    // Vị trí Conveyor hiện tại dùng cho giám sát.
    CurrentConveyorPositionMM : LREAL;
	
	CaptureConveyorPos      : REAL;     // Position conveyor lúc chụp.
	
	CaptureRobotPos         : ST_POS;   // Position robot lúc chụp.

    VisionPos               : ST_POS;   // Position vision trả về.

    // Điểm Score của Vision.
    // Với Sensor có thể gán mặc định 100%.
    VisionScore : REAL;

    // TRUE nếu góc Object có giá trị tin cậy.
    OrientationValid : BOOL;
	
// 	// TRUE khi Object Vision đã có kết quả Pose hợp lệ.
// 	VisionResultValid : BOOL;

    // TRUE khi Object đã được một Tool giữ chỗ.
    Reserved : BOOL;

    // ToolID đang giữ Object.
    ReservedToolID : UINT;

    // Trạng thái Object.
    State : E_TrackingObjectState;
	
    TriggerID               : UDINT;    // TriggerID vision.
    ProductID               : UDINT;    // ID sản phẩm.

    CameraID                : UINT;     // Camera đã chụp.
    JobID                   : UINT;     // Job đã sử dụng.

    

    ConveyorOffset          : REAL;     // Conveyor dịch từ lúc chụp.
    ConveyorCoordinate      : REAL;     // Tọa độ dọc conveyor hiện tại.

    CurrentPos              : ST_POS;   // Position hiện tại của object.

    InspectionResult        : E_InspectionResult; // Kết quả kiểm tra.
    PickAttempts            : UINT;     // Số lần thử gắp.

    RejectCode              : UINT;     // Mã lý do reject.
    ErrorID                 : UDINT;    // Mã lỗi object.
	
	// TRUE khi object còn đủ thời gian và nằm trong vùng có thể nhận gắp.
    CanPick              : BOOL;

    // Thời gian ước tính còn lại trước khi tới giới hạn bắt đầu gắp, giây.
    TimeRemainingSec     : REAL;

    // TRUE khi object active đã vượt AbortPositionMM.
    AbortRequired        : BOOL;

    // Dùng debug/thống kê lý do object bị bỏ.
    MissCode             : UINT;
	// Mức ưu tiên của object.
    // Giá trị lớn hơn được ưu tiên hơn.
    Priority : UINT;

    // Điểm chất lượng kết quả Vision, thường nằm trong khoảng 0.0 đến 1.0
    // hoặc 0.0 đến 100.0 tùy phần mềm Vision.
    //VisionScore : REAL;

    // Thời gian robot ước tính cần để tiếp cận và gắp object, đơn vị giây.
    // Giai đoạn đầu có thể gán bằng cùng một giá trị cho mọi object.
    EstimatedPickTimeSec : REAL;

    // Thời điểm object được thêm vào Queue.
    // Dùng cho thuật toán FIFO.
    CaptureTime : TIME;


END_STRUCT
END_TYPE

// Just_Motion_Control_x86_64_Linux_SM_WV/Application/STRUCT_/ConveyorTracking/ST_TRACKING_QUEUE
TYPE ST_TRACKING_QUEUE :
STRUCT
    Objects             : ARRAY[0..GVL.C_MAX_TRACK_OBJECTS]
                          OF ST_TRACKING_OBJECT;

    ValidCount          : UINT;     // Tổng số object hợp lệ.
    ReservedCount       : UINT;     // Tổng số object đã reserve.

    ActiveIndex         : UINT;     // Index object đang được xử lý.
    NextObjectID        : UDINT;    // Bộ tạo ObjectID tiếp theo.

    LastResult          : E_QueueResult; // Kết quả thao tác queue gần nhất.
END_STRUCT
END_TYPE

// Just_Motion_Control_x86_64_Linux_SM_WV/Application/STRUCT_/ConveyorTracking/ST_TRACKING_RUNTIME
TYPE ST_TRACKING_RUNTIME :
STRUCT
    State               : E_TrackingState;     // Trạng thái manager.
    Request             : ST_MODULE_REQUEST;
    Response            : ST_MODULE_RESPONSE;

    SelectedObjectIndex : UINT;                // Index object đã chọn.
    SelectedObjectID    : UDINT;               // ID object đã chọn.

    ApproachPos         : ST_POS;              // Điểm approach trong PCS.
    PickPos             : ST_POS;              // Điểm pick trong PCS.
    RetractPos          : ST_POS;              // Điểm retract trong PCS.

    PCSInfo             : ST_PCS_INFO;         // Dữ liệu PCS hiện tại.

    PickSuccess         : BOOL;                // TRUE khi gắp thành công.
    ErrorInfo           : ST_ERROR_INFO;       // Thông tin lỗi.
END_STRUCT
END_TYPE

// Just_Motion_Control_x86_64_Linux_SM_WV/Application/STRUCT_/ConveyorTracking/ST_TRACKING_SIMULATION_CONFIG
TYPE ST_TRACKING_SIMULATION_CONFIG :
STRUCT
	Mode : E_ApplicationSimulationMode;

    // Encoder ảo.
    VirtualEncoderEnable : BOOL;
    VirtualEncoderReset : BOOL;
    VirtualEncoderStepPerCycle : DINT;

    // Object giả.
    FixedObjectEnable : BOOL;
    FixedObjectPosition : MC_COORD_REF;

    // Vacuum giả.
    AutoVacuumOK : BOOL;
    VacuumOKDelay : TIME;

    // Motion logic-only.
    LogicMotionDuration : TIME;

    // Cho phép dừng sau từng state để debug.
    SingleStateMode : BOOL;
    ContinueState : BOOL;

END_STRUCT
END_TYPE

// Just_Motion_Control_x86_64_Linux_SM_WV/Application/STRUCT_/ConveyorTracking/ST_TRACKING_WORKSPACE_CONFIG
TYPE ST_TRACKING_WORKSPACE_CONFIG :
STRUCT
	// Vị trí bắt đầu vùng thu nhận object, đơn vị mm.
    AcquireZoneStartMM : REAL;

    // Vị trí bắt đầu vùng được phép gắp, đơn vị mm.
    PickZoneStartMM : REAL;

    // Vị trí kết thúc vùng được phép gắp, đơn vị mm.
    PickZoneEndMM : REAL;

    // Vượt vị trí này mà chưa VacuumOK thì phải bỏ object active.
    AbortPositionMM : REAL;

    // Vượt vị trí này thì object chưa active bị EXPIRED.
    ExpirePositionMM : REAL;

//     // Khoảng cách tối thiểu mong muốn giữa hai object, đơn vị mm.
//     MinimumObjectSpacingMM : REAL;

    // Thời gian tối thiểu robot cần để thực hiện thao tác gắp, đơn vị giây.
    MinimumPickTimeSec : REAL;

    // Thời gian dự phòng an toàn, đơn vị giây.
    SafetyMarginTimeSec : REAL;
END_STRUCT
END_TYPE

// Just_Motion_Control_x86_64_Linux_SM_WV/Application/STRUCT_/ConveyorTracking/ST_TrackingObjectQueue
//=============================================================================
// DUT: TRACKING OBJECT QUEUE
//=============================================================================
TYPE ST_TrackingObjectQueue :
STRUCT

    // Danh sách Object.
    Objects : ARRAY[0..GVL.C_MAX_TRACK_OBJECTS] OF ST_TRACKING_OBJECT;

    // Số Object đang có trong Queue.
    Count : UINT;

    // Bộ đếm sinh ObjectID cho Sensor Source.
    NextObjectID : UDINT;

END_STRUCT
END_TYPE

// Just_Motion_Control_x86_64_Linux_SM_WV/Application/STRUCT_/ConveyorTracking/ST_VISION_TRACK_OBJECT_ITEM
TYPE ST_VISION_TRACK_OBJECT_ITEM :
STRUCT

    // TRUE khi Object này hợp lệ.
    Valid : BOOL;

    // Tọa độ Object do Vision trả.
    // Có thể là pixel hoặc mm tùy cấu hình Tracking Vision Source.
    Pos : ST_POS;

    // Score nhận dạng.
    Score : REAL;

    // Product Class nếu Vision có phân loại.
    // 0 = sử dụng ProductClassID mặc định của Source Config.
    ProductClassID : UINT;

    // ID do Vision cấp cho Detection nếu có.
    FeatureID : UDINT;

END_STRUCT
END_TYPE

// Just_Motion_Control_x86_64_Linux_SM_WV/Application/STRUCT_/ConveyorTracking/ST_VISION_TRACK_OBJECT_RESULT
TYPE ST_VISION_TRACK_OBJECT_RESULT :
STRUCT

    // TRUE khi toàn bộ danh sách Object hợp lệ.
    Valid : BOOL;

    // Số Object thực Vision trả.
    ObjectCount : UINT;

    // Danh sách Object.
    Objects :
        ARRAY[1..GVL.C_MAX_VISION_TRACK_OBJECTS_PER_FRAME]
        OF ST_VISION_TRACK_OBJECT_ITEM;

END_STRUCT
END_TYPE

// Just_Motion_Control_x86_64_Linux_SM_WV/Application/STRUCT_/ConveyorTracking/ST_VisionTrackingDetection
TYPE ST_VisionTrackingDetection :
STRUCT

    // Detection này hợp lệ.
    Valid : BOOL;

    // Pose raw Vision trả về.
    RawPos : ST_POS;

    // Score.
    Score : REAL;

    // Product Class do Vision trả.
    // 0 = dùng ProductClassID trong Config.
    ProductClassID : UINT;

    // Feature/Object ID nếu Vision có.
    FeatureID : UDINT;

END_STRUCT
END_TYPE

// Just_Motion_Control_x86_64_Linux_SM_WV/Application/STRUCT_/ConveyorTracking/ST_VisionTrackingMultiResult
TYPE ST_VisionTrackingMultiResult :
STRUCT

    // Bộ kết quả hoàn chỉnh.
    Valid : BOOL;

    // Trigger tương ứng frame ảnh.
    TriggerID : UDINT;

    // Camera.
    CameraID : UINT;

    // Job.
    JobID : UINT;

    // Vị trí Conveyor tại đúng lúc chụp ảnh.
    CaptureConveyorPositionMM : LREAL;

    // Số Object Vision tìm thấy.
    ObjectCount : UINT;

    // Danh sách Detection.
    Objects :
        ARRAY[1..GVL.C_MAX_VISION_TRACK_OBJECTS_PER_FRAME]
        OF ST_VisionTrackingDetection;

END_STRUCT
END_TYPE

// Just_Motion_Control_x86_64_Linux_SM_WV/Application/STRUCT_/ConveyorTracking/ST_VisionTrackingSourceConfig
//=============================================================================
// DUT: ST_VisionTrackingSourceConfig
//-----------------------------------------------------------------------------
// Cấu hình một nguồn Vision dùng để tạo Object cho Conveyor Tracking.
// Đây là BẢN THAY THẾ cho DUT hiện tại: giữ toàn bộ field cũ và bổ sung phần
// BACKGROUND TRIGGER ở cuối.
//=============================================================================
TYPE ST_VisionTrackingSourceConfig :
STRUCT

    //=========================================================================
    // SOURCE IDENTITY
    //=========================================================================
    Enable : BOOL;                          // TRUE = cho phép Source hoạt động.
    VisionSourceID : UINT;                  // ID duy nhất của nguồn Vision Tracking.
    VisionSourceName : STRING[32];          // Tên hiển thị trên HMI/debug.
    CameraID : UINT;                        // Camera dùng cho Source này.
    JobID : UINT;                           // Job Vision dùng để tìm Object.

    //=========================================================================
    // PRODUCT / FILTER
    //=========================================================================
    ProductClassID : UINT;                  // Class mặc định nếu Vision trả ProductClassID = 0.
    MinimumScore : REAL;                    // Object có Score thấp hơn giá trị này sẽ bị loại.
    MaxObjectCount : UINT;                  // Số Object tối đa nhận từ một frame.

    //=========================================================================
    // SCALE VISION
    //-------------------------------------------------------------------------
    // ResultInPixel = TRUE:
    //     X/Y raw của Vision được đổi pixel -> mm bằng MMPerPixelX/Y.
    // ResultInPixel = FALSE:
    //     X/Y được coi là mm; nên đặt MMPerPixelX/Y = 1.0 để dễ theo dõi.
    //=========================================================================
    ResultInPixel : BOOL;
    MMPerPixelX : REAL;
    MMPerPixelY : REAL;

    //=========================================================================
    // VISION OFFSET
    //-------------------------------------------------------------------------
    // Fine offset sau khi kết quả Vision đã được chuẩn hóa về Conveyor CS.
    // Không dùng field này thay cho Tool PickOffset hoặc Product Height.
    //=========================================================================
    VisionOffset : ST_POS;

    //=========================================================================
    // DUPLICATE FILTER
    //-------------------------------------------------------------------------
    // Dùng để so Object mới với Object đang có trong Tracking Queue.
    // Object RESERVED/TRACKING/PICKING vẫn phải được xét duplicate vì Camera
    // có thể nhìn lại đúng Object đang được Robot xử lý.
    //=========================================================================
    DuplicateToleranceXMM : REAL;
    DuplicateToleranceYMM : REAL;
    DuplicateAngleDeg : REAL;

    //=========================================================================
    // BACKGROUND CAMERA TRIGGER - NEW
    //-------------------------------------------------------------------------
    // Tracking Vision không trigger trong TRK_PICK/TRK_CREATE_PCS.
    // Source này chạy nền trong thời gian TRACK_PICK session đang active.
    //=========================================================================
    AutoTrigger : BOOL;                     // TRUE = tự trigger theo quãng đường Conveyor.
    TriggerPitchMM : REAL;                  // Conveyor đi thêm bao nhiêu mm thì phát frame mới.
    TriggerOnlyWhenMoving : BOOL;           // TRUE = chỉ trigger khi Conveyor đang chạy.
    MinimumTriggerVelocityMMs : REAL;        // Ngưỡng tốc độ coi là Conveyor đang chạy.

END_STRUCT
END_TYPE

// Just_Motion_Control_x86_64_Linux_SM_WV/Application/STRUCT_/Geometry/ST_CIRCLE_2D
TYPE ST_CIRCLE_2D :
STRUCT
    CenterPos   : ST_POS;   // Tâm đường tròn.
    Radius      : REAL;     // Bán kính, mm.
    Valid       : BOOL;     // Dữ liệu hình tròn hợp lệ.
END_STRUCT
END_TYPE

// Just_Motion_Control_x86_64_Linux_SM_WV/Application/STRUCT_/Geometry/ST_LINE_2D
TYPE ST_LINE_2D :
STRUCT
    StartPos    : ST_POS;   // Điểm đầu đoạn thẳng.
    EndPos      : ST_POS;   // Điểm cuối đoạn thẳng.
    Valid       : BOOL;     // Đoạn thẳng hợp lệ.
END_STRUCT
END_TYPE

// Just_Motion_Control_x86_64_Linux_SM_WV/Application/STRUCT_/Geometry/ST_PATH_BLOCK
TYPE ST_PATH_BLOCK :
STRUCT
    Valid           : BOOL;     // Block hợp lệ.
    PathID          : UDINT;    // ID đường chạy.

    BlockIndex      : UINT;     // Số thứ tự block.
    BlockCount      : UINT;     // Tổng số block.

    StartPointIndex : UINT;     // Index điểm đầu trong toàn bộ path.
    PointCount      : UINT;     // Số điểm trong block.

    Points          : ARRAY[0..GVL.C_MAX_PATH_BLOCK_POINTS]
                      OF ST_PATH_POINT;

    Checksum        : UDINT;    // Checksum block.
END_STRUCT
END_TYPE

// Just_Motion_Control_x86_64_Linux_SM_WV/Application/STRUCT_/Geometry/ST_PATH_DATA
TYPE ST_PATH_DATA :
STRUCT
    Valid               : BOOL;     // Path hợp lệ.
    Complete            : BOOL;     // Đã nhận đầy đủ dữ liệu.
    Processed           : BOOL;     // Path đã qua xử lý.

    PathID              : UDINT;    // ID đường chạy.
    CoordSystem         : E_AppCoordSystem; // Hệ tọa độ của path.

    RawPointCount       : UINT;     // Số điểm vision trả về.
    ProcessPointCount   : UINT;     // Số điểm sau xử lý.

    ClosedPath          : BOOL;     // TRUE khi là đường khép kín.

    RawPoints           : ARRAY[0..GVL.C_MAX_RAW_PATH_POINTS]
                          OF ST_PATH_POINT;

    ProcessPoints       : ARRAY[0..GVL.C_MAX_PROCESS_PATH_POINTS]
                          OF ST_PATH_POINT;
END_STRUCT
END_TYPE

// Just_Motion_Control_x86_64_Linux_SM_WV/Application/STRUCT_/Geometry/ST_PATH_POINT
TYPE ST_PATH_POINT :
STRUCT
    Valid           : BOOL;                 // Điểm được sử dụng.
    Index           : UINT;                 // Thứ tự điểm.

    Pos             : ST_POS;               // Tọa độ X/Y/Z/A.
    SegmentType     : E_PathSegmentType;    // Kiểu đoạn dẫn tới điểm này.

    GlueOn          : BOOL;                 // TRUE khi cần mở keo trên đoạn.
    Speed           : REAL;                 // Tốc độ đoạn, mm/s.
    Flow            : REAL;                 // Lưu lượng keo.
    BlendRadius     : REAL;                 // Bán kính blend, mm.

    FeatureID       : UINT;                 // ID đoạn vision trả về.
END_STRUCT
END_TYPE

// Just_Motion_Control_x86_64_Linux_SM_WV/Application/STRUCT_/Glue/ST_GLUE_CONFIG
TYPE ST_GLUE_CONFIG :
STRUCT
    Enable                  : BOOL;     // Cho phép chức năng bôi keo.
    RunMode                 : E_GlueRunMode; // Chế độ chạy.

    DefaultSpeed            : REAL;     // Tốc độ mặc định, mm/s.
    DefaultFlow             : REAL;     // Lưu lượng mặc định.

    MinPointDistance        : REAL;     // Khoảng cách điểm nhỏ nhất, mm.
    MaxPointDistance        : REAL;     // Khoảng cách điểm lớn nhất, mm.

    SmoothingEnable         : BOOL;     // Cho phép làm mượt path.
    SmoothingFactor         : REAL;     // Hệ số làm mượt 0...1.

    ApproachHeight          : REAL;     // Độ cao tiếp cận, mm.
    RetractHeight           : REAL;     // Độ cao rút lên, mm.

    PreFlowTime             : TIME;     // Thời gian mở keo trước.
    PostFlowTime            : TIME;     // Thời gian giữ keo cuối path.

    GlueOutput              : UINT;     // Output điều khiển van keo.
END_STRUCT
END_TYPE

// Just_Motion_Control_x86_64_Linux_SM_WV/Application/STRUCT_/Glue/ST_GLUE_RUNTIME
TYPE ST_GLUE_RUNTIME :
STRUCT
    State               : E_GlueState;      // Trạng thái Glue Manager.
    ProcessState        : E_PathProcessState; // Trạng thái xử lý path.

    Request             : ST_MODULE_REQUEST;
    Response            : ST_MODULE_RESPONSE;

    Path                : ST_PATH_DATA;     // Path hiện tại.
    CurrentPointIndex   : UINT;             // Điểm đang được thực hiện.

    GlueOutputState     : BOOL;             // Trạng thái output keo.
    DryRun              : BOOL;             // TRUE khi không bật keo thật.

    ErrorInfo           : ST_ERROR_INFO;    // Thông tin lỗi.
END_STRUCT
END_TYPE

// Just_Motion_Control_x86_64_Linux_SM_WV/Application/STRUCT_/HMI/MainMC
TYPE MainMC :
STRUCT
	Start, Stop, Reset, Man_or_Auto : BOOL;
	yStart, yStop : BOOL;
	yLamp_Yellow, yLamp_Red, yLamp_Green, yBuzz : BOOL;
	AllwayON : BOOL := TRUE;
	AllwayOFF : BOOL := FALSE;
	
	Project_Run : BYTE; // 0 -255 project _0 none
	Mode_Run : BYTE; // 0-255 mode
	Check_Project : BOOL;
	Result_check : BYTE; // 0-none 1 ok 2 nG 3 waiting
	
	Enable_Dynamics_Limit : BOOL;
END_STRUCT
END_TYPE

// Just_Motion_Control_x86_64_Linux_SM_WV/Application/STRUCT_/HMI/MODBUS
TYPE MODBUS :
STRUCT
	en : BOOL;
	iniID : BYTE;
	port	: WORD;
	TCP_UDP	: BOOL;
	DelayRespTime : WORD;
END_STRUCT
END_TYPE

// Just_Motion_Control_x86_64_Linux_SM_WV/Application/STRUCT_/HMI/Project
TYPE Project :
STRUCT
	Project_Run : BYTE; // 0 -255 project _0 none
	Mode_Run : BYTE; // 0-255 mode
	
END_STRUCT
END_TYPE

// Just_Motion_Control_x86_64_Linux_SM_WV/Application/STRUCT_/HMI/TimeRun
TYPE TimeRun :
STRUCT
	Run, Stop , Wait , CLEAR : BOOL;
	Run_S, Run_M, Run_H,
	Stop_S, Stop_M, Stop_H,
	Wait_S, Wait_M, Wait_H,
	Total_S, Total_M, Total_H : WORD;
END_STRUCT
END_TYPE

// Just_Motion_Control_x86_64_Linux_SM_WV/Application/STRUCT_/Modbus/ST_VISION_MODBUS_CONTROL
TYPE ST_VISION_MODBUS_CONTROL :
STRUCT
    RunCalib : BOOL;                                // ControlWord bit2: yêu cầu chạy Calibration.
    CalibPosReady : BOOL;                           // ControlWord bit3: 12 điểm Calibration đã sẵn sàng.
    AckResult : BOOL;                               // ControlWord bit4: PLC đã nhận toàn bộ Result.
    AckBlock : BOOL;                                // ControlWord bit5: PLC đã đọc xong Block hiện tại.
    CalibPointCount : UINT;                         // Số điểm Calibration hợp lệ, tối đa 12.
    RequestBlockIndex : UINT;                       // Block tiếp theo PLC yêu cầu Vision nạp.
    AckBlockIndex : UINT;                           // Block PLC vừa đọc xong.
    CommandCode : UINT;                             // Dự phòng cho Manual/Calibration command.
    CalibrationPoints : ARRAY[1..12] OF ST_POS;     // Chỉ dùng X/Y/A trong mapping Modbus.
END_STRUCT
END_TYPE

// Just_Motion_Control_x86_64_Linux_SM_WV/Application/STRUCT_/Modbus/ST_VISION_MODBUS_STATUS
TYPE ST_VISION_MODBUS_STATUS :
STRUCT
    HeartBeat : BOOL;                               // StatusWord bit0.
    TriggerDone : BOOL;                             // StatusWord bit1.
    CalibDone : BOOL;                               // StatusWord bit2.
    ResultReady : BOOL;                             // StatusWord bit3.
    Busy : BOOL;                                    // StatusWord bit4.
    Run1Slot : BOOL;                                // StatusWord bit5.
    BlockReady : BOOL;                              // StatusWord bit6.
    Error : BOOL;                                   // StatusWord bit7.
    CalibBusy : BOOL;                               // StatusWord bit8.
    CalibError : BOOL;                              // StatusWord bit9.
    BlockIndex : UINT;                              // Block hiện tại trong MultiDataBuffer.
    BlockDataCount : UINT;                          // Số record thực trong Block.
END_STRUCT
END_TYPE

// Just_Motion_Control_x86_64_Linux_SM_WV/Application/STRUCT_/MOTOR/MOTOR_DATA
TYPE MOTOR_DATA :
STRUCT
	POS : ARRAY[0..50] OF REAL;
	SPEED_HIGH, SPEED_MID, SPEED_LOW : REAL;

	MOTION_ACC, MOTION_DEC, MOTION_JERK : REAL;
	LinearDistanceJog, AngularDistanceJog : REAL;
	Fac_Vel, Fac_Acc, Fac_Jerk,Fac_Torque : REAL;
	
	LIMIT_FW, LIMIT_BW: REAL;
END_STRUCT
END_TYPE

// Just_Motion_Control_x86_64_Linux_SM_WV/Application/STRUCT_/MOTOR/MOTOR_IN
TYPE MOTOR_IN :
STRUCT
	Power, Enable, Reset,
	Auto, Manual, Lock,
	HOME, 
	JOG_FW, JOG_BW : BOOL;
	Comfirm_Move, Comfirm_Teach: BOOL;
	LIMIT_FW, LIMIT_BW : LREAL;
	SPEED, ACC, DEC, JERK : REAL;
	Control_w_speed, Control_w_mode : WORD;
END_STRUCT
END_TYPE

// Just_Motion_Control_x86_64_Linux_SM_WV/Application/STRUCT_/MOTOR/MOTOR_OUT
TYPE MOTOR_OUT :
STRUCT
	Ready, Runing, Pause, Stop, 
	ERROR, SAFETY_CHECK : BOOL;
	M_Homed : BOOL;
	CUR_POS: REAL;
	CUR_SP : REAL;
END_STRUCT
END_TYPE

// Just_Motion_Control_x86_64_Linux_SM_WV/Application/STRUCT_/Project/Data_Point_Calib
TYPE Data_Point_Calib :
STRUCT	
	X_POS : ARRAY[0..50] OF REAL;
	Y_POS : ARRAY[0..50] OF REAL;
	Z_POS : ARRAY[0..50] OF REAL;
	R_POS : ARRAY[0..50] OF REAL;
END_STRUCT
END_TYPE

// Just_Motion_Control_x86_64_Linux_SM_WV/Application/STRUCT_/Project/Data_Project_3
TYPE Data_Project_3 :
STRUCT	
	Trigger_Auto, Trigger_Man, Trigger : BOOL; // on chup Cam
	Enable_RB_B, Enable_RB_A : BOOL;
	Shape_T1, Shape_T2 : WORD;
	Data_PlaceB_PickA, Data_PlaceA : ARRAY[0..3] OF WORD;
	
	AllowRB_In_TableC, AllowRB_In_TableA, AllowRB_In_TableB  : WORD; // =0 None : = 1: Allow_RB_B_Place , =2 :Allow_RB_A_Pick 
	
	Pro_A, Pro_B : WORD;
	NextStep_A, NextStep_B, Auto_Man_A, Auto_Man_B : BOOL;
END_STRUCT
END_TYPE

// Just_Motion_Control_x86_64_Linux_SM_WV/Application/STRUCT_/Project/Data_Project
TYPE Data_Project :
STRUCT
	Model_RB_A : ARRAY [0..10] OF Model_Data_RB;
	Model_RB_B : ARRAY [0..10] OF Model_Data_RB;
END_STRUCT
END_TYPE

// Just_Motion_Control_x86_64_Linux_SM_WV/Application/STRUCT_/Project/Project_2
TYPE Project_2 :
STRUCT
	P1,P2,P3,P4 : WORD; // địa chỉ pos
	
	P1_Z,P2_Z,P3_Z,P4_Z : WORD; // số lượng z
	
	pitchZ1, pitchZ2, pitchZ3, pitchZ4 : REAL; // khoảng cách z
	
	P1_Z_,P2_Z_,P3_Z_,P4_Z_  :WORD; // monitor
	
END_STRUCT
END_TYPE

// Just_Motion_Control_x86_64_Linux_SM_WV/Application/STRUCT_/Project/Project_3
TYPE Project_3 :
STRUCT
	
	P1,P2,P3,P4 : WORD; // địa chỉ pos
	
	P1_Z,P2_Z,P3_Z,P4_Z : WORD; // số lượng z
	
	pitchZ1, pitchZ2, pitchZ3, pitchZ4 : REAL; // khoảng cách z
	Delay_T1, Delay_T2 : WORD; 
	
	P1_Z_,P2_Z_,P3_Z_,P4_Z_  :WORD; // monitor
	Target_T1, Target_T2 : ST_POS;
	
	
END_STRUCT
END_TYPE

// Just_Motion_Control_x86_64_Linux_SM_WV/Application/STRUCT_/Project/Project_3_VISION
TYPE Project_3_VISION :
STRUCT
	vis_1, vis_2 : WORD; // địa chỉ pos
	
	Pos_vision_T1, Pos_vision_T1_Offset : ST_POS;
	Pos_vision_T2, Pos_vision_T2_Offset : ST_POS;
	
	Pos_No_T1, Pos_No_T2 : WORD;
	Number_trigger_False : WORD;
	Delay_T1, Delay_T2 : WORD;
	
	Pos_Target_T1, Pos_Target_T2 : ST_POS;
	Status_T1, Status_T2 :WORD;
	
END_STRUCT
END_TYPE

// Just_Motion_Control_x86_64_Linux_SM_WV/Application/STRUCT_/ROBOT/Model_Data_RB_ALL
TYPE Model_Data_RB_ALL :
STRUCT
	DATA_RB_A: RB_DATA;
	DATA_RB_B: RB_DATA;
	Model_Name: STRING[20];
END_STRUCT
END_TYPE

// Just_Motion_Control_x86_64_Linux_SM_WV/Application/STRUCT_/ROBOT/Model_Data_RB
TYPE Model_Data_RB :
STRUCT
	DATA_RB: RB_DATA;
	Model_Name: STRING[20];
END_STRUCT
END_TYPE

// Just_Motion_Control_x86_64_Linux_SM_WV/Application/STRUCT_/ROBOT/Move_Point
TYPE Move_Point :
STRUCT
	Enable	  : BOOL;
	Hand_Type : INT; // o: Trai-A; 1: Phai-B
	Move_Type : INT; // 0: MovP ; 1-MovL; 2-MovC
	A_Error   : BOOL;
	B_Error   : BOOL;
END_STRUCT
END_TYPE

// Just_Motion_Control_x86_64_Linux_SM_WV/Application/STRUCT_/ROBOT/Move_Type
{attribute 'qualified_only'}
{attribute 'strict'}
TYPE Move_Type :
(
	Move_P := 0,
	Move_L := 1,
	Move_C := 2
);
END_TYPE

// Just_Motion_Control_x86_64_Linux_SM_WV/Application/STRUCT_/ROBOT/PCS_Data
TYPE PCS_Data :
STRUCT
	P1_Old, P2_Old, P3_Old, P_Transform, P1_New, P2_New, P3_New : Pos_Coordsystem;
END_STRUCT
END_TYPE

// Just_Motion_Control_x86_64_Linux_SM_WV/Application/STRUCT_/ROBOT/Pos_Coordsystem
TYPE Pos_Coordsystem :
STRUCT
	X , Y , Z, A, B , C : REAL;
END_STRUCT
END_TYPE

// Just_Motion_Control_x86_64_Linux_SM_WV/Application/STRUCT_/ROBOT/Project_And_Model
TYPE Project_And_Model :
STRUCT
	Project_No_Current : INT;
	Model_No_Current : INT;
	Direction_Robot_Current : INT; // huong robot: 0-thuan; 1: nguoc
END_STRUCT
END_TYPE

// Just_Motion_Control_x86_64_Linux_SM_WV/Application/STRUCT_/ROBOT/RB_DATA
TYPE RB_DATA :
STRUCT
	X_POS : ARRAY[0..500] OF REAL;
	Y_POS : ARRAY[0..500] OF REAL;
	Z_POS : ARRAY[0..500] OF REAL;
	R_POS : ARRAY[0..500] OF REAL;
	
	SPEED_HIGH, SPEED_MID, SPEED_LOW : REAL;
	SPEED_FAC_HIGH, SPEED_FAC_MID, SPEED_FAC_LOW : REAL;

	SPEED_HIGH_MAN, SPEED_MID_MAN, SPEED_LOW_MAN : REAL;
	
	MOTION_ACC, MOTION_DEC, MOTION_JERK : REAL;
	MOTION_ACC_MAN, MOTION_DEC_MAN, MOTION_JERK_MAN : REAL;

	LinearDistanceJog, AngularDistanceJog, DistanceInchingJog : REAL;
	
	LIMIT_X_FW, LIMIT_X_BW,LIMIT_Y_FW, LIMIT_Y_BW,LIMIT_Z_FW, LIMIT_Z_BW,LIMIT_R_FW, LIMIT_R_BW : REAL;
	
	LIMIT_M1_FW, LIMIT_M1_BW,LIMIT_M2_FW, LIMIT_M2_BW,LIMIT_M3_FW, LIMIT_M3_BW,LIMIT_M4_FW, LIMIT_M4_BW : REAL;
	
	ENABLE_SOFT_LIMIT : BOOL;
	
	Fac_Vel, Fac_Acc, Fac_Jerk,Fac_Torque : REAL;
	MAX_VEL, MAX_ACC, MAX_JERK, MAX_TOQUE : REAL;
	
	Fac_Vel_Man, Fac_Acc_Man, Fac_Jerk_Man,Fac_Torque_Man : REAL;
	
	WORK_MIN_X,WORK_MAX_X, WORK_MIN_Y,WORK_MAX_Y : REAL;
	Torque_Limit : Torque_Axis;
	RB_Working_Dir : INT;
	Coordinate_Auto : ARRAY[0..100] OF INT; // Dung cho cac diem
	Data_Tranform : ARRAY [0..10] OF PCS_Data;
	
END_STRUCT
END_TYPE

// Just_Motion_Control_x86_64_Linux_SM_WV/Application/STRUCT_/ROBOT/RB_IN
TYPE RB_IN :
STRUCT
	Power, Enable, Reset,
	
	M1, M2, M3, M4,
	BK1, BK2, BK3, BK4,
	Auto, Manual, Lock,
	ORG_M1,ORG_M2,ORG_M3,ORG_M4, HOME, 
	M1_goHome, M2_goHome, M3_goHome, M4_goHome,
	ABC_as_ACS,
	RB_goHome_Comfirm,
	Home_Free_All, Home_Lock_All,
	JOG_X_FW, JOG_X_BW, 
	JOG_Y_FW, JOG_Y_BW,
	JOG_Z_FW, JOG_Z_BW,
	JOG_R_FW, JOG_R_BW,
	
	Comfirm_Move, Comfirm_Up_Z, Comfirm_Up_Z_XY_BF_R, Comfirm_Up_Z_R_BF_XY, Comfirm_Teach,
	Jog_continue, Jog_Inching, Jog_Point,
	
	Move_Z_Wait, Move_XY_Wait, Move_R_Wait,
	move_Pos_cam					 : BOOL;
	
	Number_Tool : WORD;
	ss_vacuum_1, ss_vacuum_2 : BOOL;
	Vacuum_1, Vacuum_2 : BOOL;
	
	DEL_ALL_DATA_POS : BOOL;
	
	COORD: SMC_COORD_SYSTEM;
	Control_w_speed, Control_w_mode : WORD;
	
	SPEED, ACC, DEC, JERK : REAL;
END_STRUCT
END_TYPE

// Just_Motion_Control_x86_64_Linux_SM_WV/Application/STRUCT_/ROBOT/RB_IN_Man
TYPE RB_IN_Man :
STRUCT
	SPEED_High_Man, SPEED_Mid_Man, SPEED_Low_Man, ACC_Man, DEC_Man, JERK_Man, FacVel_Man, FacAcc_Man, Fac_Dec_Man, Fac_Jerk_Man: REAL;
END_STRUCT
END_TYPE

// Just_Motion_Control_x86_64_Linux_SM_WV/Application/STRUCT_/ROBOT/RB_OUT
TYPE RB_OUT :
STRUCT
	Ready, Runing, Pause, Stop, 
	ERROR, SAFETY_CHECK : BOOL;
	M1_Homed, M2_Homed, M3_Homed, M4_Homed : BOOL;
	
	CUR_X, CUR_Y, CUR_Z, CUR_R : REAL;
	CUR_SP_X, CUR_SP_Y, CUR_SP_Z, CUR_SP_R : REAL;
	
	Tool_1, Tool_2 : BOOL; // 0 : không có hàng, 1 có hàng
END_STRUCT
END_TYPE

// Just_Motion_Control_x86_64_Linux_SM_WV/Application/STRUCT_/ROBOT/RB_Signal_Input
TYPE RB_Signal_Input :
STRUCT
	SS_DOG_Z_RIGHT_RBB, SS_DOG_Z_LEFT_RBA, Door_Sensor, Interlock, HMI_START, HMI_EMG, HMI_RESET, HMI_STOP : BOOL;
	SS_RBA_Tool_1, SS_RBA_Tool_2, SS_RBB_Tool_1, SS_RBB_Tool_2 : TON;
END_STRUCT
END_TYPE

// Just_Motion_Control_x86_64_Linux_SM_WV/Application/STRUCT_/ROBOT/RB_Speed_Point
TYPE RB_Speed_Point :
STRUCT
	Vel_Pos : ARRAY[0..50] OF REAL;
END_STRUCT
END_TYPE

// Just_Motion_Control_x86_64_Linux_SM_WV/Application/STRUCT_/ROBOT/ST_Condition
TYPE ST_Condition :
STRUCT
    Enable : BOOL;
    Name   : STRING[20];
    Row    : ARRAY[0..10] OF ST_ConditionRow;
    Result : BOOL;
    Error  : BOOL;
END_STRUCT
END_TYPE

// Just_Motion_Control_x86_64_Linux_SM_WV/Application/STRUCT_/ROBOT/ST_ConditionLine
TYPE ST_ConditionLine :
STRUCT
	Enable    : BOOL;
    VarType   : INT;
    Index     : INT;
    Compare   : INT;
    Value     : LREAL;
    LogicNext : INT;
END_STRUCT
END_TYPE

// Just_Motion_Control_x86_64_Linux_SM_WV/Application/STRUCT_/ROBOT/ST_ConditionRow
TYPE ST_ConditionRow :
STRUCT
    Enable   : BOOL;
    Source   : INT;       // 0=None, 1=DI, 2=DO, 3=REG, 4=VAR, 5=TIMER, 6=VISION
    Index    : INT;       // Số DI/DO/REG/VAR...
    Operator : INT;       // 1 =, 2 <>, 3 >, 4 >=, 5 <, 6 <=
    SetValue : DINT;
    LinkNext : INT;       // 0=END, 1=AND, 2=OR
    //Note     : STRING[20];
END_STRUCT
END_TYPE

// Just_Motion_Control_x86_64_Linux_SM_WV/Application/STRUCT_/ROBOT/ST_ConditionTable
TYPE ST_ConditionTable : // Struct 1 bảng điều kiện, 1 bảng có tối đa 5 dòng.
STRUCT
	Enable : BOOL;
    Name   : STRING[30];

    Row    : ARRAY[0..5] OF ST_ConditionRow;

    Result : BOOL;       // Kết quả cuối cùng
    Error  : BOOL;
END_STRUCT
END_TYPE

// Just_Motion_Control_x86_64_Linux_SM_WV/Application/STRUCT_/ROBOT/ST_MotionParam
TYPE ST_MotionParam :
STRUCT
    Speed : LREAL;
    Acc   : LREAL;
    Dec   : LREAL;
    Jerk  : LREAL;

    VelFac  : LREAL;
    AccFac  : LREAL;
    DecFac  : LREAL;
    JerkFac : LREAL;
END_STRUCT
END_TYPE

// Just_Motion_Control_x86_64_Linux_SM_WV/Application/STRUCT_/ROBOT/ST_MotionQueueItem
TYPE ST_MotionQueueItem :
STRUCT
    Cmd        : E_RobotCmd; // Lệnh Motion: MovP, MovL, MovC
    SourceStep : INT;        // Step gốc để debug lỗi

    PointNo    : INT;        // Point dùng cho MovP / MovL
    MidPointNo : INT;        // Point giữa cho MovC
    EndPointNo : INT;        // Point cuối cho MovC

    Speed : LREAL;           // Speed override, =0 thì dùng Set Speed hiện hành

    BlendMode   : INT;       // 0=None, 1=TMCornerDistance, 2=TMStartVelocity
    BlendRadius : LREAL;     // TransitionParameter[0]

    CircleMode : INT;        // Dùng cho MovC
    PathChoice : INT;        // Dùng cho MovC
	SkipPositionCheck : BOOL; // Xac dinh co check vi tri co dinh khong
	
	//==================== MEMBER MỚI ====================
    // TRUE: bỏ PointNo và sử dụng DirectPosition.
    UseDirectPosition : BOOL;

    // Tọa độ động do Application tạo ra.
    DirectPosition : ST_POS;

    // Hệ tọa độ của DirectPosition.
    DirectCoordSystem : SMC_COORD_SYSTEM;

    // Dynamic riêng. Giá trị <= 0 dùng thông số chung hiện tại.
    Acceleration : LREAL;
    Deceleration : LREAL;
    Jerk : LREAL;

    // ID nguồn để Application đối chiếu Done/Error.
    ApplicationCommandID : UDINT;
	
END_STRUCT
END_TYPE

// Just_Motion_Control_x86_64_Linux_SM_WV/Application/STRUCT_/ROBOT/ST_RobotProgram
TYPE ST_RobotProgram  :
STRUCT
	Name       : STRING[30];
	Model      : ARRAY[0..10] OF Model_Data_RB_ALL;
    StepCount_A  : INT;
    CondCount_A  : INT;
	StepCount_B  : INT;
    CondCount_B  : INT;
    Step_A       : ARRAY[0..500] OF ST_RobotStep;
    Condition_A  : ARRAY[0..100] OF ST_Condition;
	
	Point_Name_A : ARRAY[0..500] OF STRING[20];
	Step_B       : ARRAY[0..500] OF ST_RobotStep;
    Condition_B  : ARRAY[0..100] OF ST_Condition;
	//Model_B      : ARRAY[0..10] OF Model_Data_RB;
	Point_Name_B : ARRAY[0..500] OF STRING[20];
END_STRUCT
END_TYPE

// Just_Motion_Control_x86_64_Linux_SM_WV/Application/STRUCT_/ROBOT/ST_RobotStep
TYPE ST_RobotStep :
STRUCT
	GroupCmd : INT;
	Cmd     : E_RobotCmd;
    P1      : INT;
    P2      : INT;
    P3      : DINT;
    P4      : INT;
    P5      : INT;
    P6      : INT;
    P7      : INT;
    P8      : INT;
    P9      : INT;
    P10     : INT;
    P11     : INT;
    P12     : INT;
    Note    : STRING[20];
END_STRUCT
END_TYPE

// Just_Motion_Control_x86_64_Linux_SM_WV/Application/STRUCT_/ROBOT/ST_ScaraTransformDeg
TYPE ST_ScaraTransformDeg :
STRUCT
	CosT     : REAL;
    SineT     : REAL;
    ThetaDeg : REAL;

    Dx       : REAL;
    Dy       : REAL;
    Dz       : REAL;

    DeltaR   : REAL;

    Valid    : BOOL;
    Error    : BOOL;
    ErrorID  : INT;
END_STRUCT
END_TYPE

// Just_Motion_Control_x86_64_Linux_SM_WV/Application/STRUCT_/ROBOT/Torque_Axis
TYPE Torque_Axis :
STRUCT
	A0,A1,A2,A3,B0,B1,B2,B3 : INT;
END_STRUCT
END_TYPE

// Just_Motion_Control_x86_64_Linux_SM_WV/Application/STRUCT_/TOOL/ST_MultiToolTrackingCommand
//=============================================================================
// DUT: MULTI-TOOL TRACKING COMMAND
//=============================================================================
TYPE ST_MultiToolTrackingCommand :
STRUCT

    // Giữ TRUE trong suốt thời gian chạy lệnh.
    Execute : BOOL;

    // Reset application.
    Reset : BOOL;

    // Abort application.
    Abort : BOOL;

    // ID command.
    CommandID : UDINT;

    // Recipe cần chạy.
    RecipeID : UINT;

    // 0 = dùng TargetPickCount trong Recipe.
    TargetPickCountOverride : UINT;

    // 0 = dùng ToolEnableMask trong Recipe.
    ToolMaskOverride : DWORD;

END_STRUCT
END_TYPE

// Just_Motion_Control_x86_64_Linux_SM_WV/Application/STRUCT_/TOOL/ST_MultiToolTrackingRecipe
//=============================================================================
// DUT: MULTI-TOOL TRACKING RECIPE
//=============================================================================
TYPE ST_MultiToolTrackingRecipe :
STRUCT

    // Cho phép Recipe.
    Enable : BOOL;

    // ID Recipe.
    RecipeID : UINT;

    // Tên Recipe.
    RecipeName : STRING[32];

    // Nguồn Object.
    ObjectSourceType : E_ObjectSourceType;

	// Nguồn Vision cần sử dụng.
	// 0 = không lọc Source nếu anh muốn giữ chế độ wildcard.
	VisionSourceID : UINT;

    // Vision Job nếu dùng Vision.
    VisionJobID : UINT;

    // Sensor Source nếu dùng Sensor.
    SensorSourceID : UINT;

    // Bitmask các Tool được phép sử dụng.
    ToolEnableMask : DWORD;

    // Số sản phẩm cần gắp trong một lệnh TRACK_ON.
    TargetPickCount : UINT;

    // Cho phép Done khi chưa đủ số lượng nhưng đã có ít nhất một sản phẩm.
    AllowPartialPick : BOOL;

    // Product Class cần gắp.
    // 0 = tất cả.
    ProductClassID : UINT;
	
	// Cao độ mặt cần hút của sản phẩm tính từ Object reference/conveyor plane.
    // Đơn vị: mm.
    PickSurfaceHeightMM : REAL;

    // Score Vision tối thiểu.
    MinimumVisionScore : REAL;


    // Timeout chờ Object.
    ObjectWaitTimeout : TIME;

    // Timeout toàn chu trình.
    TotalTrackingTimeout : TIME;

END_STRUCT
END_TYPE

// Just_Motion_Control_x86_64_Linux_SM_WV/Application/STRUCT_/TOOL/ST_MultiToolTrackingStatus
//=============================================================================
// DUT: MULTI-TOOL TRACKING STATUS
//=============================================================================
TYPE ST_MultiToolTrackingStatus :
STRUCT

    // Xung báo đã nhận lệnh.
    Accepted : BOOL;

    // Application đang chạy.
    Busy : BOOL;

    // Application hoàn thành.
    Done : BOOL;

    // Application lỗi.
    Error : BOOL;

    // Mã lỗi.
    ErrorID : UDINT;

    // CommandID vừa xử lý.
    ResponseCommandID : UDINT;

    // State hiện tại.
    State : E_MultiTrackState;

    // Recipe đang chạy.
    ActiveRecipeID : UINT;

    // Tool đang được chọn.
    SelectedToolID : UINT;

    // Object đang được chọn.
    SelectedObjectID : UDINT;

    // Số sản phẩm đã gắp.
    PickedCount : UINT;

    // Số sản phẩm yêu cầu.
    TargetPickCount : UINT;

    // Bitmask Tool đang giữ sản phẩm.
    OccupiedToolMask : DWORD;

    // Tracking Core đã đồng bộ.
    TrackingSyncOK : BOOL;

    // PCS hiện đang InUse.
    PCSInUse : BOOL;

END_STRUCT
END_TYPE

// Just_Motion_Control_x86_64_Linux_SM_WV/Application/STRUCT_/TOOL/ST_ToolCommand
//=============================================================================
// DUT: TOOL COMMAND
//=============================================================================
TYPE ST_ToolCommand :
STRUCT

    // Xung Execute của lệnh.
    Execute : BOOL;

    // Reset Tool.
    Reset : BOOL;

    // Abort Tool.
    Abort : BOOL;

    // ID của lệnh.
    CommandID : UDINT;

    // Tool cần điều khiển.
    ToolID : UINT;

    // Action cần chạy.
    CommandType : E_ToolCommandType;

    // ObjectID liên quan tới lệnh Grip.
    ObjectID : UDINT;

END_STRUCT
END_TYPE

// Just_Motion_Control_x86_64_Linux_SM_WV/Application/STRUCT_/TOOL/ST_ToolConfig
//=============================================================================
// DUT: TOOL CONFIG
//=============================================================================
TYPE ST_ToolConfig :
STRUCT

    // Cho phép Tool.
    Enable : BOOL;

    // Cho phép Tool được sử dụng trong Tracking.
    AllowTracking : BOOL;

    // ID duy nhất của Tool.
    ToolID : UINT;

    // Tên hiển thị trên HMI.
    ToolName : STRING[32];

    // Loại Tool.
    ToolType : E_ToolType;

    // TCP thực tế đã hiệu chuẩn so với Flange.
    ToolTCP : ST_POS;

    // Offset gắp riêng của Tool so với Object Frame.
    PickOffset : ST_POS;

    // Độ cao Approach riêng của Tool.
    ApproachHeight : REAL;

    // TRUE nếu Tool có cơ cấu Up/Down độc lập.
    UseUpDown : BOOL;
	// Hành trình cơ khí từ vị trí UP xuống vị trí DOWN, đơn vị mm.
	UpDownStroke : REAL;
    // Cấu hình IO.
    IO : ST_ToolIOConfig;

    // Thời gian giả lập Down OK nếu không có DI.
    DownTimeNoSensor : TIME;

    // Thời gian giả lập Up OK nếu không có DI.
    UpTimeNoSensor : TIME;

    // Thời gian giả lập Grip OK nếu không có DI.
    GripTimeNoSensor : TIME;

    // Thời gian thực hiện Release nếu không có DI.
    ReleaseTimeNoSensor : TIME;

    // Timeout Down.
    DownTimeout : TIME;

    // Timeout Up.
    UpTimeout : TIME;

    // Timeout Grip.
    GripTimeout : TIME;

    // Timeout Release.
    ReleaseTimeout : TIME;

    // Delay xác nhận Grip OK ổn định.
    GripConfirmDelay : TIME;

    // Độ ưu tiên của Tool.
    Priority : UINT;

    // Product Class mà Tool được phép gắp.
    // 0 = cho phép tất cả.
    AllowedProductClassID : UINT;

END_STRUCT
END_TYPE

// Just_Motion_Control_x86_64_Linux_SM_WV/Application/STRUCT_/TOOL/ST_ToolIOConfig
//=============================================================================
// DUT: TOOL IO CONFIG
//-----------------------------------------------------------------------------
// Tất cả kênh IO đều dùng chỉ số logic.
// Channel = 0 nghĩa là không sử dụng kênh đó.
//=============================================================================
TYPE ST_ToolIOConfig :
STRUCT

    // TRUE = Up/Down dung chung mot DO.
    // FALSE = Down va Up dung hai DO doc lap.
    UseSingleUpDownDO : BOOL;

    // DO dung chung khi UseSingleUpDownDO = TRUE.
    // Channel = 0 nghia la khong su dung.
    UpDownDOChannel : UINT;

    // Hai DO doc lap khi UseSingleUpDownDO = FALSE.
    DownDOChannel : UINT;
    UpDOChannel : UINT;
	
	// TRUE = Up/Down dung chung mot DO.
    // FALSE = Down va Up dung hai DO doc lap.
    UseSingleGripReleaseDO  : BOOL;

    // DO dung chung khi UseSingleGripReleaseDO = TRUE.
    // Channel = 0 nghia la khong su dung.
    GripReleaseDOChannel : UINT;


    // Grip / Release.
    GripDOChannel : UINT;
    ReleaseDOChannel : UINT;

    // Feedback DI.
    DownOKDIChannel : UINT;
    UpOKDIChannel : UINT;
    GripOKDIChannel : UINT;
    PartPresentDIChannel : UINT;

    // Active level.
    // Single DO mode:
    //   DOWN = DownDOActiveLevel
    //   UP   = NOT DownDOActiveLevel
    DownDOActiveLevel : BOOL;

    // Chi dung trong Dual DO mode.
    UpDOActiveLevel : BOOL;

    GripDOActiveLevel : BOOL;
    ReleaseDOActiveLevel : BOOL;
    DownOKDIActiveLevel : BOOL;
    UpOKDIActiveLevel : BOOL;
    GripOKDIActiveLevel : BOOL;
    PartPresentDIActiveLevel : BOOL;

END_STRUCT
END_TYPE

// Just_Motion_Control_x86_64_Linux_SM_WV/Application/STRUCT_/TOOL/ST_ToolStatus
//=============================================================================
// DUT: TOOL STATUS
//=============================================================================
TYPE ST_ToolStatus :
STRUCT

    // Xung báo đã nhận lệnh.
    Accepted : BOOL;

    // Tool đang thực thi lệnh.
    Busy : BOOL;

    // Xung báo lệnh hoàn thành.
    Done : BOOL;

    // Tool báo lỗi.
    Error : BOOL;

    // Mã lỗi.
    ErrorID : UDINT;

    // CommandID vừa xử lý.
    ResponseCommandID : UDINT;

    // ToolID của Status.
    ToolID : UINT;

    // State hiện tại của Tool.
    State : E_ToolRuntimeState;

    // Phản hồi Tool Up.
    UpOK : BOOL;

    // Phản hồi Tool Down.
    DownOK : BOOL;

    // Phản hồi Grip.
    GripOK : BOOL;

    // Phản hồi có sản phẩm.
    PartPresent : BOOL;

    // TRUE khi Tool đang giữ sản phẩm.
    Occupied : BOOL;

    // ObjectID đang được giữ.
    HeldObjectID : UDINT;

END_STRUCT
END_TYPE

// Just_Motion_Control_x86_64_Linux_SM_WV/Application/STRUCT_/Vision/ST_ALIGN_CONFIG
TYPE ST_ALIGN_CONFIG :
STRUCT
    Enable          : BOOL;             // Cho phép chức năng align.
    MinScore        : REAL;             // Score nhỏ nhất được chấp nhận.

    MaxOffsetX      : REAL;             // Độ lệch X tối đa, mm.
    MaxOffsetY      : REAL;             // Độ lệch Y tối đa, mm.
    MaxOffsetZ      : REAL;             // Độ lệch Z tối đa, mm.
    MaxOffsetA      : REAL;             // Độ lệch góc tối đa, độ.

    CameraToRobot   : ST_Transform2D;  // Transform camera sang robot.
END_STRUCT
END_TYPE

// Just_Motion_Control_x86_64_Linux_SM_WV/Application/STRUCT_/Vision/ST_ALIGN_RESULT
TYPE ST_ALIGN_RESULT :
STRUCT
    Valid           : BOOL;         // Kết quả align hợp lệ.
    RawOffset       : ST_POS;       // Offset trực tiếp từ vision.
    RobotOffset     : ST_POS;       // Offset sau khi đổi sang hệ robot.
    Score           : REAL;         // Score nhận dạng.
    FeatureID       : UINT;         // Đặc trưng đã nhận dạng.
END_STRUCT
END_TYPE

// Just_Motion_Control_x86_64_Linux_SM_WV/Application/STRUCT_/Vision/ST_ALIGN_RUNTIME
TYPE ST_ALIGN_RUNTIME :
STRUCT
    State           : E_AlignState;     // Trạng thái Align Manager.
    Request         : ST_MODULE_REQUEST;
    Response        : ST_MODULE_RESPONSE;

    Result          : ST_ALIGN_RESULT;  // Kết quả align hiện tại.
    WorkOffset      : ST_Transform2D;  // Work offset đang được áp dụng.

    ErrorInfo       : ST_ERROR_INFO;    // Thông tin lỗi align.
END_STRUCT
END_TYPE

// Just_Motion_Control_x86_64_Linux_SM_WV/Application/STRUCT_/Vision/ST_AlignResult
TYPE ST_AlignResult :
STRUCT
	Valid       : BOOL;    // TRUE khi kết quả align hợp lệ.
    Offset      : ST_POS;  // Độ lệch X/Y/Z/A vision tìm được.
    Score       : REAL;    // Điểm tin cậy của kết quả.
    FeatureID   : UINT;    // ID đặc trưng được nhận dạng.
END_STRUCT
END_TYPE

// Just_Motion_Control_x86_64_Linux_SM_WV/Application/STRUCT_/Vision/ST_ControlWord_VS
TYPE ST_ControlWord_VS :
STRUCT
	HeartBeat : BOOL;
	TriggerCam : BOOL;
	RunCalib : BOOL;
	CalibPosReady : BOOL;
	AckResult : BOOL;
	AckBlock : BOOL;
	ResetVision : BOOL;
	AbortVision : BOOL;
END_STRUCT
END_TYPE

// Just_Motion_Control_x86_64_Linux_SM_WV/Application/STRUCT_/Vision/ST_INSPECTION_CONFIG
TYPE ST_INSPECTION_CONFIG :
STRUCT
    Enable          : BOOL;     // Cho phép chức năng inspection.
    RetryEnable     : BOOL;     // Cho phép chụp lại khi lỗi.
    MaxRetry        : UINT;     // Số lần chụp lại tối đa.

    FailAsError     : BOOL;     // TRUE: sản phẩm NG được coi là lỗi hệ thống.
    RejectOutput    : UINT;     // Ngõ ra điều khiển cơ cấu reject.
END_STRUCT
END_TYPE

// Just_Motion_Control_x86_64_Linux_SM_WV/Application/STRUCT_/Vision/ST_INSPECTION_ITEM
TYPE ST_INSPECTION_ITEM :
STRUCT
    ItemID          : UINT;     // ID hạng mục kiểm tra.
    Valid           : BOOL;     // Dữ liệu hạng mục hợp lệ.
    ResultOK        : BOOL;     // TRUE khi hạng mục đạt.

    DefectCode      : UINT;     // Mã loại khuyết tật.
    Score           : REAL;     // Score phát hiện lỗi.

    MeasuredValue   : REAL;     // Giá trị đo được.
    MinLimit        : REAL;     // Giới hạn dưới.
    MaxLimit        : REAL;     // Giới hạn trên.

    DefectPos       : ST_POS;   // Vị trí khuyết tật.
    DefectWidth     : REAL;     // Chiều rộng khuyết tật, mm.
    DefectHeight    : REAL;     // Chiều cao khuyết tật, mm.
END_STRUCT
END_TYPE

// Just_Motion_Control_x86_64_Linux_SM_WV/Application/STRUCT_/Vision/ST_INSPECTION_RESULT
TYPE ST_INSPECTION_RESULT :
STRUCT
    Valid           : BOOL;                 // Toàn bộ kết quả hợp lệ.
    OverallOK       : BOOL;                 // Kết quả tổng thể PASS/FAIL.
    Result          : E_InspectionResult;   // Trạng thái kết quả.

    ItemCount       : UINT;                 // Số hạng mục thực tế.
    FailCount       : UINT;                 // Số hạng mục không đạt.

    Items           : ARRAY[0..GVL.C_MAX_INSPECTION_ITEMS]
                      OF ST_INSPECTION_ITEM;
END_STRUCT
END_TYPE

// Just_Motion_Control_x86_64_Linux_SM_WV/Application/STRUCT_/Vision/ST_INSPECTION_RUNTIME
TYPE ST_INSPECTION_RUNTIME :
STRUCT
    State           : E_InspectionState;    // Trạng thái Inspection Manager.
    Request         : ST_MODULE_REQUEST;
    Response        : ST_MODULE_RESPONSE;

    Result          : ST_INSPECTION_RESULT; // Kết quả kiểm tra.
    RetryCount      : UINT;                 // Số lần đã chụp lại.

    ErrorInfo       : ST_ERROR_INFO;        // Thông tin lỗi.
END_STRUCT
END_TYPE

// Just_Motion_Control_x86_64_Linux_SM_WV/Application/STRUCT_/Vision/ST_InspectionItem
TYPE ST_InspectionItem  :
STRUCT
	ItemID          : UINT;    // ID hạng mục kiểm tra.

    Valid           : BOOL;    // TRUE khi dữ liệu hợp lệ.
    ResultOK        : BOOL;    // TRUE khi hạng mục đạt.

    DefectCode      : UINT;    // Mã lỗi khuyết tật.
    Score           : REAL;    // Điểm tin cậy.

    MeasuredValue   : REAL;    // Giá trị đo được.
    MinLimit        : REAL;    // Giới hạn dưới.
    MaxLimit        : REAL;    // Giới hạn trên.

    DefectPos       : ST_POS;  // Vị trí lỗi.
    DefectWidth     : REAL;    // Chiều rộng lỗi, mm.
    DefectHeight    : REAL;    // Chiều cao lỗi, mm.
END_STRUCT
END_TYPE

// Just_Motion_Control_x86_64_Linux_SM_WV/Application/STRUCT_/Vision/ST_PathPoint
TYPE ST_PathPoint  :
STRUCT
	Valid           : BOOL;                // Điểm có được sử dụng hay không.
    Index           : UINT;                // Thứ tự điểm.

    Pos             : ST_POS;              // Tọa độ điểm X/Y/Z/A.

    SegmentType     : E_PathSegmentType;   // Loại đoạn dẫn tới điểm này.
    GlueOn          : BOOL;                // TRUE khi cần bật keo.

    Speed           : REAL;                // Tốc độ tại đoạn này, mm/s.
    Flow            : REAL;                // Lưu lượng keo.
    BlendRadius     : REAL;                // Bán kính blend, mm.

    FeatureID       : UINT;                // ID đoạn hoặc đặc trưng vision.
END_STRUCT
END_TYPE

// Just_Motion_Control_x86_64_Linux_SM_WV/Application/STRUCT_/Vision/ST_StatusWord_VS
TYPE ST_StatusWord_VS :
STRUCT
	HeartBeat : BOOL;
	TriggerDone : BOOL;
	CalibDone : BOOL;
	ResultReady : BOOL;
	Busy : BOOL;
	Run1Slot : BOOL;
	BlockReady : BOOL;
	Error : BOOL;
	CalibBusy : BOOL;
	CalibError : BOOL;
END_STRUCT
END_TYPE

// Just_Motion_Control_x86_64_Linux_SM_WV/Application/STRUCT_/Vision/ST_TrayConfig
//=============================================================================
// DUT: ST_TrayConfig
//-----------------------------------------------------------------------------
// Chỉ teach một MasterPos; các slot khác được tính bằng pitch local của Tray.
//=============================================================================
TYPE ST_TrayConfig :
STRUCT
    Enable : BOOL;
    TrayID : UINT;
    MasterPosID : UINT;                     // PositionID của slot tham chiếu.
    RowCount : UINT;
    ColumnCount : UINT;
    RowPitchMM : REAL;
    ColumnPitchMM : REAL;
    FillByRow : BOOL;                       // TRUE = đi theo hàng trước, FALSE = theo cột trước.
END_STRUCT
END_TYPE

// Just_Motion_Control_x86_64_Linux_SM_WV/Application/STRUCT_/Vision/ST_TrayRuntime
//=============================================================================
// DUT: ST_TrayRuntime
//=============================================================================
TYPE ST_TrayRuntime :
STRUCT
    CurrentIndex : UINT;                    // Slot tiếp theo cần đặt, bắt đầu từ 1.
    FilledCount : UINT;
    Full : BOOL;
END_STRUCT
END_TYPE

// Just_Motion_Control_x86_64_Linux_SM_WV/Application/STRUCT_/Vision/ST_VISION_ALIGN_REQUEST
TYPE ST_VISION_ALIGN_REQUEST :

STRUCT

    //=========================================================================

    // COMMAND - dữ liệu Robot gửi sang Vision Manager

    //=========================================================================

    Execute : BOOL;                  // TRUE = Robot yêu cầu bắt đầu/duy trì transaction Vision.

    CameraID : UINT;                 // Camera/Vision Channel cần sử dụng.

    JobID : UINT;                    // Job Vision cần chạy trên Camera.


    //=========================================================================

    // STATUS - Vision Manager trả về cho Robot

    //=========================================================================

    Busy : BOOL;                     // TRUE = Request đã được Manager nhận và đang xử lý.

    Done : BOOL;                     // TRUE = Transaction kết thúc bình thường, đã có business result.

    Error : BOOL;                    // TRUE = Lỗi communication/protocol/configuration/timeout.

    ErrorID : INT;                   // Mã lỗi Manager hoặc lỗi chuyển tiếp từ FB_VisionAlign.


    //=========================================================================

    // BUSINESS RESULT - kết quả dùng cho logic chương trình Robot

    //=========================================================================

    ResultOK : BOOL;                 // TRUE = VIS_RESULT_OK; FALSE = NG/NOT_FOUND/LOW_SCORE/...

    ResultValid : BOOL;              // Cờ Valid của dữ liệu Vision.

    ResultStatus : E_VisionResultStatus; // Trạng thái business result từ Vision.


    //=========================================================================

    // RESULT DATA - dữ liệu Vision đã chốt của transaction

    //=========================================================================

    TriggerID : UDINT;               // TriggerID của transaction vừa hoàn thành.

    X : REAL;                        // Kết quả X.

    Y : REAL;                        // Kết quả Y.

    Z : REAL;                        // Kết quả Z.

    A : REAL;                        // Kết quả góc A.

    Score : REAL;                    // Điểm Score.

    FeatureID : UINT;                // Feature/Object ID do Vision trả về.

END_STRUCT

END_TYPE

// Just_Motion_Control_x86_64_Linux_SM_WV/Application/STRUCT_/Vision/ST_VISION_CHANNEL_STATUS
TYPE ST_VISION_CHANNEL_STATUS :
STRUCT
    Enable              : BOOL;                 // Camera được bật hay không.
    Online              : BOOL;                 // Kết nối camera đang hoạt động.
    Ready               : BOOL;                 // Vision sẵn sàng nhận lệnh.
    Busy                : BOOL;                 // Vision đang xử lý ảnh.
    ResultReady         : BOOL;                 // Kết quả đã sẵn sàng.

    State               : E_VisionState;        // State hiện tại của kênh.
    ResultStatus        : E_VisionResultStatus; // Trạng thái kết quả.

    CurrentJobID        : UINT;                 // Job đang chạy.
    CurrentTriggerID    : UDINT;                // TriggerID đang xử lý.

    RetryCount          : UINT;                 // Số lần đã thử lại.
    Error               : BOOL;                 // Kênh đang có lỗi.
    ErrorID             : UDINT;                // Mã lỗi.
END_STRUCT
END_TYPE

// Just_Motion_Control_x86_64_Linux_SM_WV/Application/STRUCT_/Vision/ST_VISION_COMMAND
TYPE ST_VISION_COMMAND :
STRUCT
    Execute             : BOOL;                 // Bắt đầu lệnh vision.
    Abort               : BOOL;                 // Hủy lệnh đang chạy.
    Reset               : BOOL;                 // Reset kênh vision.

    CameraID            : UINT;                 // Camera thực hiện lệnh.
    JobID               : UINT;                 // Job vision cần chạy.
    Application         : E_VisionApplication;  // Loại ứng dụng.

    TriggerID           : UDINT;                // ID ghép lệnh và kết quả.
    ProductID           : UDINT;                // ID sản phẩm.

    CaptureRobotPos     : ST_POS;               // Vị trí robot lúc chụp.
    CaptureConveyorPos  : REAL;                 // Vị trí conveyor lúc chụp, mm.
END_STRUCT
END_TYPE

// Just_Motion_Control_x86_64_Linux_SM_WV/Application/STRUCT_/Vision/ST_VISION_CONFIG
TYPE ST_VISION_CONFIG :
STRUCT
    Enable              : BOOL;     // Cho phép sử dụng camera.
    SimulationMode      : BOOL;     // TRUE khi dùng dữ liệu mô phỏng.

    CameraID            : UINT;     // ID camera.
	
	Robot : E_VisionRobot;    // Tay Robot được phép sử dụng Camera này.
	
    BaseAddress         : UINT;     // Địa chỉ Modbus bắt đầu của camera.

    CommandOffset       : UINT;     // Offset vùng lệnh PLC gửi vision.
    StatusOffset        : UINT;     // Offset vùng trạng thái vision.
    HeaderOffset        : UINT;     // Offset vùng header kết quả.
    DataOffset          : UINT;     // Offset vùng dữ liệu kết quả.

    PositionScale       : REAL;     // Hệ số chuyển dữ liệu vị trí thành mm.
    AngleScale          : REAL;     // Hệ số chuyển dữ liệu góc thành độ.
    ScoreScale          : REAL;     // Hệ số chuyển score thô thành giá trị thực.

    TriggerTimeout      : TIME;     // Thời gian tối đa chờ vision nhận trigger.
    ResultTimeout       : TIME;     // Thời gian tối đa chờ kết quả.
    BlockTimeout        : TIME;     // Thời gian tối đa chờ một block dữ liệu.

    MaxPointCount       : UINT;     // Số điểm tối đa camera được phép trả.
    MaxRetry            : UINT;     // Số lần chụp lại tối đa.

    CameraToRobot       : ST_Transform2D;
    // Phép biến đổi từ hệ tọa độ camera sang hệ robot.
	
END_STRUCT
END_TYPE

// Just_Motion_Control_x86_64_Linux_SM_WV/Application/STRUCT_/Vision/ST_VISION_JOB_CONFIG
TYPE ST_VISION_JOB_CONFIG :
STRUCT
    Enable              : BOOL;                 // Cho phép sử dụng job.
    CameraID            : UINT;                 // Camera chứa job.
    JobID               : UINT;                 // Số job trên phần mềm vision.
    Application         : E_VisionApplication;  // Loại ứng dụng của job.
    ExpectedDataType    : E_VisionDataType;     // Kiểu payload dự kiến.

    MinScore            : REAL;                 // Score nhỏ nhất được chấp nhận.
    MaxResultCount      : UINT;                 // Số kết quả tối đa.

    PositionLimitX      : ST_RANGE_REAL;        // Giới hạn tọa độ X.
    PositionLimitY      : ST_RANGE_REAL;        // Giới hạn tọa độ Y.
    PositionLimitZ      : ST_RANGE_REAL;        // Giới hạn tọa độ Z.
    AngleLimitA         : ST_RANGE_REAL;        // Giới hạn góc A.
END_STRUCT
END_TYPE

// Just_Motion_Control_x86_64_Linux_SM_WV/Application/STRUCT_/Vision/ST_VISION_POS_RESULT
TYPE ST_VISION_POS_RESULT :
STRUCT
    Valid       : BOOL;     // TRUE khi tọa độ hợp lệ.
    Pos         : ST_POS;   // Tọa độ X/Y/Z/A do vision trả về.
    Score       : REAL;     // Điểm tin cậy.
    FeatureID   : UINT;     // ID đặc trưng hoặc mẫu.
END_STRUCT
END_TYPE

// Just_Motion_Control_x86_64_Linux_SM_WV/Application/STRUCT_/Vision/ST_VISION_RESULT
TYPE ST_VISION_RESULT :
STRUCT

    Header : ST_VISION_RESULT_HEADER;

    // Một Pose.
    PosResult : ST_VISION_POS_RESULT;

    // N Object độc lập dùng cho Conveyor Tracking.
    TrackObjectResult : ST_VISION_TRACK_OBJECT_RESULT;

    AlignResult : ST_ALIGN_RESULT;

    Inspection : ST_INSPECTION_RESULT;

    PathID : UDINT;

    PathValid : BOOL;

END_STRUCT
END_TYPE

// Just_Motion_Control_x86_64_Linux_SM_WV/Application/STRUCT_/Vision/ST_VISION_RESULT_HEADER
TYPE ST_VISION_RESULT_HEADER :
STRUCT
    Valid : BOOL;                                   // TRUE khi Result hoàn chỉnh.
    CameraID : UINT;                                // Camera trả Result.
    JobID : UINT;                                   // Job đã chạy.
    Application : E_VisionApplication;              // Loại ứng dụng.
    DataType : E_VisionDataType;                    // Kiểu payload.
    TriggerID : UDINT;                              // Ghép command/result.
    ProductID : UDINT;                              // Product ID nếu dùng.
    ResultStatus : E_VisionResultStatus;            // OK/NG/NotFound/Error...
    ResultCode : UINT;                              // Mã Result phía Vision.
    ErrorCode : UINT;                               // Mã lỗi phía Vision.
    DataCount : UINT;                               // Tổng record của Result.
    BlockCount : UINT;                              // Tổng số Block.
    BlockIndex : UINT;                              // Block hiện tại/Block cuối đã decode.
    BlockDataCount : UINT;                          // Số record thực trong Block.
    Checksum : UDINT;                               // Optional.
    CaptureConveyorPos : REAL;                      // Encoder lúc chụp.
END_STRUCT
END_TYPE

// Just_Motion_Control_x86_64_Linux_SM_WV/Application/STRUCT_/Vision/ST_VisionAlignRecipe
//=============================================================================
// DUT: ST_VisionAlignRecipe
//=============================================================================
TYPE ST_VisionAlignRecipe :
STRUCT
    Enable : BOOL;
    RecipeID : UINT;
    CameraID : UINT;                        // Camera dùng để Align.
    JobID : UINT;                           // Job Align.
    ToolCount : UINT;                       // Số Tool tham gia Recipe.
    Tools : ARRAY[1..GVL.C_MAX_TOOLS] OF ST_VisionAlignToolConfig;
END_STRUCT
END_TYPE

// Just_Motion_Control_x86_64_Linux_SM_WV/Application/STRUCT_/Vision/ST_VisionAlignToolConfig
//=============================================================================
// DUT: ST_VisionAlignToolConfig
//-----------------------------------------------------------------------------
// Cấu hình iterative alignment cho từng Tool.
// CaptureMasterPosID là điểm bắt đầu Align; các lần chụp tiếp theo KHÔNG cần
// CapturePos cố định vì Robot sẽ di chuyển theo correction của lần trước.
//=============================================================================
TYPE ST_VisionAlignToolConfig :
STRUCT
    Enable : BOOL;                          // Tool có tham gia Align Recipe hay không.
    ToolID : UINT;                          // Tool đang giữ sản phẩm.
    CaptureMasterPosID : UINT;              // PositionID điểm bắt đầu chụp/căn.

    MaxAlignIterations : UINT;              // Số vòng Measure -> Correct tối đa.
    ToleranceX : REAL;                      // Sai số X đạt yêu cầu, mm.
    ToleranceY : REAL;                      // Sai số Y đạt yêu cầu, mm.
    ToleranceA : REAL;                      // Sai số góc đạt yêu cầu, degree.

    MaxCorrectionX : REAL;                  // Giới hạn correction X cho một vòng.
    MaxCorrectionY : REAL;                  // Giới hạn correction Y cho một vòng.
    MaxCorrectionA : REAL;                  // Giới hạn correction A cho một vòng.
END_STRUCT
END_TYPE

// Just_Motion_Control_x86_64_Linux_SM_WV/Application/STRUCT_/Vision/ST_VisionAlignToolRuntime
//=============================================================================
// DUT: ST_VisionAlignToolRuntime
//-----------------------------------------------------------------------------
// Runtime riêng từng Tool để kết quả Tool 2 không ghi đè Tool 1.
//=============================================================================
TYPE ST_VisionAlignToolRuntime :
STRUCT
    Valid : BOOL;
    ToolID : UINT;
    Iteration : UINT;
    AlignDone : BOOL;

    LastTriggerID : UDINT;
    LastVisionResult : ST_POS;              // X/Y/A Vision của lần đo gần nhất.
    LastCorrection : ST_POS;                // Correction đã tính cho lần gần nhất.
    LastScore : REAL;
END_STRUCT
END_TYPE

// Just_Motion_Control_x86_64_Linux_SM_WV/Application/STRUCT_/Vision/ST_VisionCommand
TYPE ST_VisionCommand  :
STRUCT
	Execute             : BOOL;                // Bắt đầu yêu cầu vision.
    Abort               : BOOL;                // Hủy yêu cầu đang chạy.
    Reset               : BOOL;                // Reset lỗi và trạng thái FB.

    CameraID            : UINT;                // Camera được chọn.
    JobID               : UINT;                // Job vision cần chạy.
    Application         : E_VisionApplication; // Loại ứng dụng vision.

    TriggerID           : UDINT;               // ID dùng ghép lệnh và kết quả.
    ProductID           : UDINT;               // ID sản phẩm đang xử lý.

    CaptureRobotPos     : ST_POS;              // Tọa độ robot tại lúc camera chụp.
    CaptureConveyorPos  : REAL;                // Vị trí conveyor tại lúc chụp, mm.
END_STRUCT
END_TYPE

// Just_Motion_Control_x86_64_Linux_SM_WV/Application/STRUCT_/Project/Project_4/Alarm_P_4
TYPE Alarm_P_4 :
STRUCT
	Alarm_Limit_NG_VS, Alarm_Limit_NG_TS : BOOL;
	Alarm_TS_SS_Up, Alarm_TS_NG_Pass_Fail_Signal, Alarm_VS_NG_Pass_Fail_Signal, Alarm_VS_SS_JigOut, Alarm_Limit_Test_TS, Alarm_Limit_Test_VS : BOOL;
	Wait_Product_Input, Read_Barcode_TS, Read_Barcode_VS, Full_NG_CONV : BOOL;
END_STRUCT
END_TYPE

// Just_Motion_Control_x86_64_Linux_SM_WV/Application/STRUCT_/Project/Project_4/Pro4_auto
TYPE Pro4_auto :
STRUCT
	TS_On_Off,
	Vs_On_Off,
	Trigger_Barcode_Ts_On_Off,
	Trigger_Barcode_Vs_On_Off,
	Lighting_On_Off,
	Cv_NG_On_Off,
	centering_ts_On_Off, Trigger_Vs_Align_On_Off, Run_Calib_Pos_Done 		: BOOL := FALSE;
	
	Alarm_Not_barcode, comfirm_Reduct_Pro, Alarm_Not_barcode_VS, Alarm_VS_Align, comfirm_Reduct_Pro_NG_Vs_Align : BOOL;
	NG_CV_Full_Pro : BOOL;
	signal_Ts_pass, Signal_Ts_Fail,
	signal_vs_pass, Signal_Vs_fail,
	Pass_Barcode_ts, Pass_Barcode_vs : BOOL;
	
	Result_Trigger_Vs_Align_Done, Result_Calib_Done : BOOL;
	
	D_Ts, D_Vs, D_Bar_Ts, D_Bar_vs : WORD;
	
	D_CV_NG : WORD;
	Nb_Pro_OK, Nb_Pro_NG : INT;
	T_tacktime_cr, T_tacktime_pre: INT;
	Fac_Vel_Max_A, Fac_Vel_Max_B: REAL;
	Fac_Acc_Max_A, Fac_Acc_Max_B: REAL;
	Fac_Jerk_Max_A, Fac_Jerk_Max_B: REAL;
	TORQUE_LIMIT_SET_A0, TORQUE_LIMIT_SET_A1, TORQUE_LIMIT_SET_A2, TORQUE_LIMIT_SET_A3 : INT;
	TORQUE_LIMIT_SET_B0, TORQUE_LIMIT_SET_B1, TORQUE_LIMIT_SET_B2, TORQUE_LIMIT_SET_B3 : INT;
	Nb_NG_VS_Limit, Nb_NG_TS_Limit : INT;
	
END_STRUCT
END_TYPE

// Just_Motion_Control_x86_64_Linux_SM_WV/Application/STRUCT_/Project/Project_4/Pro4_Input
TYPE Pro4_Input :
STRUCT
	T_AT1, T_AT2, T_BT1, T_BT2,
	T_Ts_Result_Scanner,
	T_Ts_Pass,
	T_Ts_Fail,
	T_Door_ss,
	T_Ts_Press_Up,
	T_Ts_Check_Gap,
	T_Vs_detect,
	T_Cv_In_1,
	T_Cv_In_2,
	T_Cv_OK_out,
	T_Vs_Result_Scanner,
	T_Vs_Pass,
	T_Vs_Fail,
	T_Cv_NG_out_1,
	T_Cv_NG_out_2,
	T_Cv_NG_out_full : TON;
	
END_STRUCT
END_TYPE

// Just_Motion_Control_x86_64_Linux_SM_WV/Application/STRUCT_/Project/Project_4/Pro4_manual
TYPE Pro4_manual :
STRUCT
	TS_On_Off,
	Vs_On_Off,
	Trigger_Barcode_Ts_On_Off,
	Trigger_Barcode_Vs_On_Off,
	Lighting_On_Off,
	Cv_NG_On_Off,
	centering_ts_On_Off, Trigger_Vs_Align_On_Off, Run_Calib_Pos_Done, Run_Calib_Pos, Result_Trigger_Vs_Align_Done, Result_Calib_Done : BOOL := FALSE;
	
	signal_Ts_pass, Signal_Ts_Fail,
	signal_vs_pass, Signal_Vs_fail,
	Pass_Barcode_ts, Pass_Barcode_vs : BOOL;
	
	D_Ts, D_Vs, D_Bar_Ts, D_Bar_vs : WORD;
	
END_STRUCT
END_TYPE

// Just_Motion_Control_x86_64_Linux_SM_WV/Application/STRUCT_/Project/Project_4/Pro4_Monitor
TYPE Pro4_Monitor :
STRUCT
	D_Day_Pro, D_Night_Pro : ARRAY[0..11] OF WORD;
	D_Day_Pro_OK, D_Night_Pro_OK : ARRAY[0..11] OF WORD;
	D_Day_Pro_NG_VS, D_Night_Pro_NG_VS : ARRAY[0..11] OF WORD;
	D_Day_Pro_NG_TS, D_Night_Pro_NG_TS : ARRAY[0..11] OF WORD;
	Total_Day, Total_Night, All_Shift : WORD;
	Total_Day_OK, Total_Night_OK, All_Shift_OK : WORD;
	Total_Day_NG, Total_Night_NG, All_Shift_NG : WORD;
	Total_Day_NG_VS, Total_Night_NG_VS, All_Shift_NG_VS : WORD;
	Total_Day_NG_TS, Total_Night_NG_TS, All_Shift_NG_TS : WORD;
	
END_STRUCT
END_TYPE

// Just_Motion_Control_x86_64_Linux_SM_WV/Application/STRUCT_/Project/Project_4/Pro4_Process
TYPE Pro4_Process :
STRUCT
	NextStep_B, NextStep_A : BOOL;
	Re_Trigger_Barcode_Ts, Re_Trigger_Barcode_Vs, Re_Trigger_VS_Align : BOOL;
	Device_Process_A, Device_Process_B :WORD;
	
	DATA_TOOL_A1_IN, DATA_TOOL_A2_OUT, DATA_TOOL_A1_IN_OLD, DATA_TOOL_A2_OUT_OLD,
	DATA_TOOL_B1_IN, DATA_TOOL_B1_IN_OLD : WORD;
	
	DATA_MC_TS, DATA_MC_VS : WORD;
	
	Clear_Data : BOOL;
	
	Pos_vision_T2_Offset, Pos_vision_T1_Offset : ST_POS;
	
	Pos_Target_T1, Pos_Target_T2 : ST_POS;
END_STRUCT
END_TYPE

// Just_Motion_Control_x86_64_Linux_SM_WV/Application/STRUCT_/Project/Project_4/Pro4_RB_Pos
TYPE Pro4_RB_Pos :
STRUCT
	Wait,BF_Pick_T1, Pick_T1, Barcode_T1, 
		BF_Pick_T2, Pick_T2,
		BF_Place_T1_OK, Place_T1_Ok,
		BF_Place_T1_NG, Place_T1_NG,
		BF_Place_T2_OK, Place_T2_Ok,
		BF_Place_T2_NG, Place_T2_NG : BOOL;
	
	
END_STRUCT
END_TYPE

// Just_Motion_Control_x86_64_Linux_SM_WV/Application/STRUCT_/Project/Project_4/Pro4_setting
TYPE Pro4_setting :
STRUCT
	TDelay_pick_T1, TDelay_pick_T2,
	TDelay_Place_T1, Tdelay_Place_T2 : WORD;
	
END_STRUCT
END_TYPE

// Just_Motion_Control_x86_64_Linux_SM_WV/Application/STRUCT_/Project/Project_4/Pro4_Setting_Funtion
TYPE Pro4_Setting_Funtion :
STRUCT
	Delay_Trigger_Barcode_Ts : WORD;
	Delay_Trigger_Barcode_Vs : WORD;
	
	Mode_Dry, Mode_Auto_Pass_TS, Mode_Auto_Pass_Vs,
	Mode_Skip_Barcode_ts, Mode_Skip_Barcode_vs,
	Mode_Skip_ss_T1_A,
	Mode_Skip_ss_T2_A,
	Mode_Skip_ss_T1_b, Mode_ByPass_TS, Mode_Skip_VS_Align : BOOL;
	Delay_Trigger_Vision_Align : WORD;
	
END_STRUCT
END_TYPE

// Just_Motion_Control_x86_64_Linux_SM_WV/Application/STRUCT_/Project/Project_4/Project4
TYPE Project4 :
STRUCT
	RB_A, RB_B : Pro4_RB_Pos;
	Auto : Pro4_auto;
	Man : Pro4_manual;
	ST_A, ST_B : Pro4_setting;
	ST_MC : Pro4_Setting_Funtion ;
	Signal_In : Pro4_Input;
	Process : Pro4_Process;
	Monitor : Pro4_Monitor;
END_STRUCT
END_TYPE

// Just_Motion_Control_x86_64_Linux_SM_WV/Application/GVL_1
{attribute 'qualified_only'}
VAR_GLOBAL PERSISTENT
	DATA_RB_B: RB_DATA;
	DATA_RB_A: RB_DATA;
	Point_Name_A    : ARRAY [0..500] OF STRING[20];
	Name_Program_Cr : STRING[30];
    StepCount_Cr_A  : INT;
    CondCount_Cr_A  : INT;
    Step_Cr_A       : ARRAY[0..500] OF ST_RobotStep;
    Condition_Cr_A  : ARRAY[0..100] OF ST_Condition;
	Point_Name_B    : ARRAY [0..500] OF STRING[20];
    StepCount_Cr_B  : INT;
    CondCount_Cr_B  : INT;
    Step_Cr_B       : ARRAY[0..500] OF ST_RobotStep;
    Condition_Cr_B  : ARRAY[0..100] OF ST_Condition;
	//A_CondTable : ARRAY[0..100] OF ST_Condition;

    A_Reg : ARRAY[0..200] OF DINT;
    A_Var : ARRAY[0..200] OF DINT;
	B_Reg : ARRAY[0..200] OF DINT;
    B_Var : ARRAY[0..200] OF DINT;
	
// 	// Cấu hình từng Tool.
//     g_aToolConfigA : ARRAY[0..GVL.C_MAX_TOOLS] OF ST_ToolConfig;
// 
//     // Cấu hình các nguồn Sensor.
//     g_aSensorSourceConfigA : ARRAY[0..8] OF ST_SensorObjectSourceConfig;
// 
//     // Tracking Recipe.
//     g_aMultiTrackRecipeA : ARRAY[0..32] OF ST_MultiToolTrackingRecipe;


END_VAR

// Just_Motion_Control_x86_64_Linux_SM_WV/Application/GLOBAL_/GVL_2
{attribute 'qualified_only'}
VAR_GLOBAL RETAIN	
	Project1_RB_A_Get, Project1_RB_A_Put, Project1_RB_B_Get, Project1_RB_B_Put : Pallets_In;
	Project1_RB_A_Get_, Project1_RB_A_Put_, Project1_RB_B_Get_, Project1_RB_B_Put_  : Pallets_Out;
END_VAR

VAR_GLOBAL RETAIN	
	
	Project2_RB_A_Get, Project2_RB_A_Put, Project2_RB_B_Get, Project2_RB_B_Put : Project_2;
	
	pro3_B_get : Project_3_VISION;
	Pro3_B_Put, Pro3_A_Get, Pro3_A_Put : Project_3;
	Process3 : Data_Project_3;
END_VAR

VAR_GLOBAL RETAIN
	A_Tool : ARRAY[0..4] OF Pos_Coordsystem;
	B_Tool : ARRAY[0..4] OF Pos_Coordsystem;
	A_POS_COOR , B_POS_COOR : Pos_Coordsystem;
	
END_VAR

// Just_Motion_Control_x86_64_Linux_SM_WV/Application/GLOBAL_/GVL
{attribute 'qualified_only'}
VAR_GLOBAL
	//DEFIND INPUT ROBOT
	MB_ : ARRAY[0..1000] OF BOOL; // 
	Alarm_ : ARRAY[0..500] OF BOOL;
	DW_ : ARRAY[0..100] OF WORD;
	Y : ARRAY[0..100] OF BOOL; // 
	X : ARRAY[0..100] OF BOOL; // 
	MODBUS : ARRAY[0..1999] OF WORD; // AT %QW30 :
	Log_HMI : ARRAY[0..20] OF STRING(255); 
	Log_RobotA, Log_RobotB : ARRAY[0..20]  OF STRING(255); 
END_VAR

VAR_GLOBAL // CONTROL ROBOT
	RB_A, RB_B : RB_IN;
	RB_A_Man, RB_B_Man : RB_IN_Man;
	RB_A_, RB_B_ : RB_OUT;
	RBA_VEL_POS, RBB_VEL_POS : RB_Speed_Point;
	
	HMI_MAIN : MainMC;
	Cam_T1, Cam_T2 : ModbusCam;
	COOR_A_CONVERT : ARRAY[0..9] OF Pos_Coordsystem;
	COOR_B_CONVERT : ARRAY[0..9] OF Pos_Coordsystem;
	Pro4_ : Project4;
	//Pos_bonus : ARRAY[0..100] OF ST_POS;
END_VAR
// namnv3103
VAR_GLOBAL
	Fac_Vel_Set_A, Fac_Vel_Slow : REAL;
	Fac_Vel_Set_B, Fac_Acc_Set_B, Fac_Jerk_Set_B, Fac_Torque_Set_B: REAL;
	Fac_Acc_Set_A, Fac_Jerk_Set_A, Fac_Torque_Set_A: REAL;
	Torque_Max : Torque_Axis;
	Reset_Torque_Max : BOOL;
	Alarm_Robot : Alarm_Robot;
	Alarm_P4 : Alarm_P_4;
	ConfirmNG_VS, ConfirmNG_TS : BOOL := FALSE;
	Reset_Alarm_History : BOOL;
	Project_No_Cur, Model_No_Cur, RB_Direction_Cur: INT;
	ProjectAndModel : Project_And_Model; 
	Project : ARRAY[0..10] OF Data_Project;
	Project_Cur : ARRAY[0..10] OF BOOL;
	Project_Cur_Rev : ARRAY[0..10] OF BOOL;
	Save_Model, Call_Model : BOOL;
	RB_Signal_In : RB_Signal_Input;
	Data_Calib_RB : ARRAY[0..10] OF Calib_Cam_Input_Model;
	Calib_Cam_RB : ARRAY[0..10] OF Calib_Cam;
	Man_Calib_RB, Auto_VS_RB : ARRAY[0..10] OF VS_Control;
	NB_Register_Modbus_VS : INT := 150;
	Save_Data_Cam, Load_Data_Cam : ARRAY[0..10] OF BOOL;
	RTrig_Save_Data_Cam, RTrig_Load_Data_Cam : ARRAY[0..10] OF R_TRIG;
	
	
END_VAR
VAR_GLOBAL
	RB_B_Calib_Point : Data_Point_Calib;
END_VAR
VAR_GLOBAL RETAIN
	TimeMachine : TimeRun;
END_VAR

VAR_GLOBAL
	HMI_A_ViewStartStep : INT := 1;
    HMI_A_ViewStepNo    : ARRAY[0..10] OF INT;
	HMI_A_ViewGroupCmd  : ARRAY[0..10] OF INT;
    HMI_A_ViewCmd       : ARRAY[0..10] OF INT;

    HMI_A_ViewP1        : ARRAY[0..10] OF INT;
    HMI_A_ViewP2        : ARRAY[0..10] OF INT;
    HMI_A_ViewP3        : ARRAY[0..10] OF DINT;
    HMI_A_ViewP4        : ARRAY[0..10] OF INT;
    HMI_A_ViewP5        : ARRAY[0..10] OF INT;
    HMI_A_ViewP6        : ARRAY[0..10] OF INT;
    HMI_A_ViewNote      : ARRAY[0..10] OF STRING[20];

    HMI_A_RowState      : ARRAY[0..10] OF INT;
	HMI_A_RowSelect     : ARRAY[0..10] OF BOOL;
	HMI_A_RowSelectedCmd : INT;
	HMI_A_LengthRowCmd : INT;
	A_LengthStep : INT;
END_VAR

VAR_GLOBAL
    HMI_A_SelectedViewRow : INT;
    HMI_A_SelectedStepNo  : INT;

    HMI_A_ViewCmd_Scroll_Up      : BOOL;
	HMI_A_ViewCmd_Scroll_Down    : BOOL;
	HMI_A_ViewCmd_Page_Up      : BOOL;
	HMI_A_ViewCmd_Page_Down    : BOOL;
	HMI_A_ViewCmd_Go_Bot      : BOOL;
	HMI_A_ViewCmd_Go_Top    : BOOL;
	HMI_A_ViewCmd_Scroll_Up_Old      : BOOL;
	HMI_A_ViewCmd_Scroll_Down_Old    : BOOL;
	HMI_A_ViewCmd_Page_Up_Old      : BOOL;
	HMI_A_ViewCmd_Page_Down_Old    : BOOL;
	HMI_A_ViewCmd_Go_Bot_Old      : BOOL;
	HMI_A_ViewCmd_Go_Top_Old    : BOOL;
END_VAR

VAR_GLOBAL
    HMI_A_EditStepNo   : INT;
    HMI_A_EditGroupCmd : INT; // nhom lenh su dung
	HMI_A_EditCmd      : E_RobotCmd;

    HMI_A_EditP1       : INT;
    HMI_A_EditP2       : INT;
    HMI_A_EditP3       : DINT;
    HMI_A_EditP4       : INT;
    HMI_A_EditP5       : INT;
    HMI_A_EditP6       : INT;


    HMI_A_EditNote   : STRING[20];
    HMI_A_EditCmdReq : INT; //20 =  Edit, 21 = Add, 22 = Insert, 23 = Delete Step, 24 = Save Step, 25 = Copy Step, 26 = Paste Step
	HMI_A_EditCmdReq_Arr : ARRAY [0..20] OF BOOL; 
	HMI_A_EditSelgroupCmd : ARRAY [0..10] OF BOOL; // dung de enable cac phan command theo tung group
	HMI_A_Edit_Trigger_Windown_Cmd: ARRAY [0..10] OF BOOL; // dung de hien thi cac man hinh cai dat theo tham so cua chuong trinh theo tung group cmd
	HMI_A_Edit_Show_Help : BOOL; // Hien thi man hinh gia thich cac tham so
END_VAR

VAR_GLOBAL

    //========================================================
    // CLIPBOARD 1 STEP
    //========================================================
    A_StepClipboardValid : BOOL := FALSE;
    A_StepClipboard      : ST_RobotStep;   // đổi ST_Step theo đúng TYPE của Step_Cr_A[]


    //========================================================
    // CLIPBOARD NHIỀU STEP
    //========================================================
	HMI_A_CopyStartStep : INT;
	HMI_A_CopyEndStep   : INT;

    A_StepCopyStart : INT := 0;
    A_StepCopyEnd   : INT := 0;

    

    

END_VAR


VAR_GLOBAL
	Robot_Programs : ARRAY [0..20] OF ST_RobotProgram;
	// Ví dụ cho phép copy tối đa 1000 step/lần
    AB_StepBlockClipboard : ARRAY[0..1000] OF ST_RobotStep;
	// Số lượng step đã copy
    AB_StepCopyCount : INT := 0;
	AB_StepBlockClipboardValid : BOOL := FALSE;
END_VAR
// Khai bao bien lien quan cac diem hoat dong Robot (Point table)
VAR_GLOBAL
	HMI_A_PointNo        : ARRAY[0..10] OF INT;
	HMI_A_ViewStartPoint : INT := 1;
    HMI_A_View_Pos_X     : ARRAY[0..10] OF REAL;
    HMI_A_View_Pos_Y     : ARRAY[0..10] OF REAL;
    HMI_A_View_Pos_Z     : ARRAY[0..10] OF REAL;
    HMI_A_View_Pos_R     : ARRAY[0..10] OF REAL;
    HMI_A_View_Pos_Name  : ARRAY[0..10] OF STRING[20];
	HMI_A_PointViewCmd   : INT;
	HMI_A_PointNoSelected : INT;
	HMI_A_ChangeSelectedPoint : BOOL;
END_VAR

//============================================================
// POINT CLIPBOARD
// Dùng để lưu tạm dữ liệu khi Copy/Paste Point
//============================================================
VAR_GLOBAL

    // TRUE = Clipboard đang chứa dữ liệu hợp lệ
    A_PointClipboardValid : BOOL := FALSE;

    // Số Point nguồn đã Copy - chủ yếu dùng để hiển thị/debug
    A_PointClipboardSourceNo : INT := 0;

    // Dữ liệu Point đã Copy
    A_PointClipboardName : STRING[20] := '';

    A_PointClipboardX : REAL := 0.0;
    A_PointClipboardY : REAL := 0.0;
    A_PointClipboardZ : REAL := 0.0;
    A_PointClipboardR : REAL := 0.0;

END_VAR

VAR_GLOBAL
	HMI_A_Edit_PointNo   : INT;
    HMI_A_Edit_Pos_X     : REAL;
    HMI_A_Edit_Pos_Y     : REAL;
    HMI_A_Edit_Pos_Z     : REAL;
    HMI_A_Edit_Pos_R     : REAL;
    HMI_A_Edit_Pos_Name  : STRING[20];
	HMI_A_EditPointReq   : INT; 
	HMI_A_EditPointReq_Arr : ARRAY[0..10] OF BOOL;
	HMI_A_RowSelectedPoint : INT;
	HMI_A_RowSelectedPoint_Array : ARRAY[0..10] OF BOOL;
END_VAR

// Khia bao bien cho bang dieu kien dung robot A
// Biến HMI xem danh sách 10 condition/trang
VAR_GLOBAL
    HMI_A_CondViewStart : INT := 1;

    HMI_A_CondViewNo     : ARRAY[0..10] OF INT;
    HMI_A_CondViewName   : ARRAY[0..10] OF STRING[20];
    HMI_A_CondViewEnable : ARRAY[0..10] OF BOOL;
    HMI_A_CondViewResult : ARRAY[0..10] OF BOOL;

    HMI_A_CondRowSelect  : ARRAY[0..10] OF BOOL;
    HMI_A_CondSelectedNo : INT;
	HMI_A_CondSelectedCmd : INT;

    HMI_A_CondCmd_Up       : BOOL;
    HMI_A_CondCmd_Down     : BOOL;
    HMI_A_CondCmd_PageUp   : BOOL;
    HMI_A_CondCmd_PageDown : BOOL;
    HMI_A_CondCmd_GoTop    : BOOL;
    HMI_A_CondCmd_GoBot    : BOOL;
END_VAR

// Biến HMI Edit 1 condition, nhưng thấy 10 dòng điều kiện
VAR_GLOBAL
    HMI_A_CondEditNo     : INT;
    HMI_A_CondEditName   : STRING[20];
    HMI_A_CondEditEnable : BOOL;

    HMI_A_CondEditRowEnable : ARRAY[0..10] OF BOOL;
    HMI_A_CondEditSource    : ARRAY[0..10] OF INT;
    HMI_A_CondEditIndex     : ARRAY[0..10] OF INT;
    HMI_A_CondEditOperator  : ARRAY[0..10] OF INT;
    HMI_A_CondEditSetValue  : ARRAY[0..10] OF DINT;
    HMI_A_CondEditLinkNext  : ARRAY[0..10] OF INT;
    HMI_A_CondEditNote      : ARRAY[0..10] OF STRING[30];
	HMI_A_CondMonitorEnable : BOOL; // Nút Monitor ON/OFF

    HMI_A_CondMonActualValue : ARRAY[0..10] OF DINT;
    HMI_A_CondMonRowResult   : ARRAY[0..10] OF BOOL;
    HMI_A_CondMonFinalResult : BOOL;

    HMI_A_CondCmdReq : INT;
    // 1=Load, 2=Save, 3=Clear, 4=Copy, 5=Paste, 6=DeleteRow, 7=InsertRow

    HMI_A_CondEditSelectedRow : INT;
    HMI_A_CondCopied : ST_Condition;
END_VAR

////////////////////
VAR_GLOBAL
    A_CopyStepBuffer : ST_RobotStep;
    A_CopyStepValid  : BOOL;

    A_MaxStep        : INT := 1000;
    A_MaxViewStart   : INT := 991;
END_VAR

VAR_GLOBAL
    A_RunEnable    : BOOL;
    A_RunPause     : BOOL;
    A_RunStop      : BOOL;

    A_RunStep      : INT := 1;
    A_RunBusy      : BOOL;
    A_RunDone      : BOOL;
    A_RunAlarm     : BOOL;
    A_RunAlarmCode : INT;

    A_RunState     : INT := 0;
    A_StepActive   : BOOL;
	
END_VAR
// Khai bao phan tham so co the chay Blend va MovC
VAR_GLOBAL
    A_CurrentMotionParam : ST_MotionParam := (
        Speed := 500.0,
        Acc := 2000.0,
        Dec := 2000.0,
        Jerk := 10000.0,
        VelFac := 1.0,
        AccFac := 1.0,
        DecFac := 1.0,
        JerkFac := 1.0
    );

    A_MotionQueue : ARRAY[0..20] OF ST_MotionQueueItem;
    A_MotionHead  : INT := 1; // Vi tri lay du lieu o trong  Queue
    A_MotionTail  : INT := 1; // Vi tri ghi du lieu o trong Queue
    A_MotionCount : INT := 0; // So luong Motion co trong hang doi
	A_PipelineUsedCount : INT := 0; // So luong Motion da dua vao pipeline
    A_MotionQueueStart : BOOL;
    A_MotionQueueBusy  : BOOL;
    A_MotionQueueDone  : BOOL;
    A_MotionQueueError : BOOL;
    A_MotionQueueState : INT;

    A_MotionScanStep   : INT;
    A_MotionBlockEndStep : INT;

    A_MotionItemActive : ST_MotionQueueItem;
    A_MotionItemValid  : BOOL;

    A_MotionAccepted   : BOOL;
    A_MotionAllDone    : BOOL;

    A_MotionAlarmCode  : INT;
END_VAR

// PRG_A_MotionQueueBuilder
// VAR_GLOBAL
//     A_MotionManagerStart : BOOL;
//     A_MotionManagerDone  : BOOL;
//     A_MotionManagerBusy  : BOOL;
//     A_MotionManagerError : BOOL;
// END_VAR
// PRG_A_MotionManager
VAR_GLOBAL
    // Số slot motion dùng để blend
    A_MoveSlotBusy      : ARRAY[0..3] OF BOOL;
    A_MoveSlotCmd       : ARRAY[0..3] OF E_RobotCmd;
    A_MoveSlotItem      : ARRAY[0..3] OF ST_MotionQueueItem;

    A_MoveSlotStart     : ARRAY[0..3] OF BOOL;
    A_MoveSlotAccepted  : ARRAY[0..3] OF BOOL;
    A_MoveSlotDone      : ARRAY[0..3] OF BOOL;
    A_MoveSlotError     : ARRAY[0..3] OF BOOL;
    A_MoveSlotErrorID   : ARRAY[0..3] OF INT;
	A_MoveSlotReleasePending : ARRAY[0..3] OF BOOL;
    A_QueueSendFinished : BOOL;
    A_ActiveMotionCount : INT; // so luong motion dang active

    A_MotionManagerState : INT;
	
	A_MotionAbortReq  : BOOL;
    A_MotionAbortDone : BOOL;
	
	A_MotionDoneQueue : ARRAY[0..20] OF INT;

//     A_MotionDoneHead  : INT := 1;
//     A_MotionDoneTail  : INT := 1;
//     A_MotionDoneCount : INT := 0;
// 	A_MoveSlotReset : ARRAY[0..3] OF BOOL;
	
END_VAR

VAR_GLOBAL CONSTANT
	C_BM_Aborting         : INT := 0;
    C_BM_BlendingHigh     : INT := 5;
    C_BM_BlendingLow      : INT := 2;
    C_BM_BlendingNext     : INT := 4;
    C_BM_BlendingPrevious : INT := 3;
    C_BM_Buffered         : INT := 1;

    C_TM_CornerDistance   : INT := 2;
    C_TM_None             : INT := 0;
    C_TM_StartVelocity    : INT := 1;
END_VAR

VAR_GLOBAL
	MotionTolXYZ : REAL := 0.03; // Do chinh xac so sanh cho truc XYZ
	MotionTolR : REAL := 0.04;  // Do chinh xac so sanh cho truc R
END_VAR

// PRG_A_MotionQueueBuilder
VAR_GLOBAL
    A_MotionQueueSize : INT := 20;

    A_MotionStreamEnable : BOOL := TRUE;
    A_MotionStreamBusy   : BOOL;
    A_MotionStreamPause  : BOOL;

    A_WaitMotionClear    : BOOL;

    A_MotionQueueAlmostFull : BOOL;
    A_MotionQueueCanPush    : BOOL;

    A_MotionManagerBusy  : BOOL;
    A_MotionManagerDone  : BOOL;
    A_MotionManagerError : BOOL;

    //A_MotionAlarmCode : INT;
END_VAR

VAR_GLOBAL
    A_PipelineDepth        : INT := 3;
    A_PipelineActive       : BOOL;
    A_PipelineNextPushStep : INT;

    A_PushMotionReq        : BOOL;
    A_PushMotionDone       : BOOL;
    A_PushMotionError      : BOOL;
    A_PushMotionItem       : ST_MotionQueueItem;

    A_MotionDonePulse      : BOOL;
    A_MotionDoneStep       : INT;

    A_MotionErrorPulse     : BOOL;
    A_MotionErrorStep      : INT;
    A_MotionErrorCode      : INT;
	A_RunErrorStep         : INT;
	A_MotionErrorSlot	   : INT;
END_VAR

VAR_GLOBAL
    A_RunMode : INT := 0;
    // 0 = Auto
    // 1 = Step

    A_StepRunReq  : BOOL; // Nút bấm chạy 1 step từ HMI
    A_StepRunEdge : BOOL;
    A_LastStepRunReq : BOOL;

    A_StepHold : BOOL;    // TRUE = đang dừng chờ bấm step tiếp
END_VAR

VAR_GLOBAL
    // Timer user
    A_TimerStart : ARRAY[0..20] OF BOOL;
    A_TimerDone  : ARRAY[0..20] OF BOOL;
    A_TimerPT    : ARRAY[0..20] OF TIME;

    // Call stack
    A_CallStack      : ARRAY[0..20] OF INT;
    A_CallStackIndex : INT;

    // Vision
    A_VisionTriggerReq  : BOOL;
    A_VisionDone        : BOOL;
    A_VisionOK          : BOOL;
    A_VisionError       : BOOL;

    // Tracking
    A_TrackEnable       : BOOL;
    A_TrackPickReq      : BOOL;
    A_TrackPlaceReq     : BOOL;
    A_TrackPickDone     : BOOL;
    A_TrackPlaceDone    : BOOL;

    // Register/Variable
    A_Reg : ARRAY[0..200] OF DINT;
    A_Var : ARRAY[0..200] OF DINT;
END_VAR

VAR_GLOBAL CONSTANT
    // Số lượng camera tối đa mà hệ thống hỗ trợ.
    C_MAX_VISION_CHANNELS : UINT := 4;

    // Số lượng job vision tối đa lưu trong cấu hình.
    C_MAX_VISION_JOBS : UINT := 32;

    // Số lượng sản phẩm tối đa cùng tồn tại trong hàng đợi tracking.
    C_MAX_TRACK_OBJECTS : UINT := 32;

    // Số điểm thô tối đa vision có thể trả cho một đường chạy.
    C_MAX_RAW_PATH_POINTS : UINT := 500;

    // Số điểm tối đa sau khi lọc và xử lý đường chạy.
    C_MAX_PROCESS_PATH_POINTS : UINT := 500;

    // Số điểm tối đa truyền trong một block Modbus.
    C_MAX_PATH_BLOCK_POINTS : UINT := 20;

    // Số hạng mục kiểm tra tối đa trong một kết quả inspection.
    C_MAX_INSPECTION_ITEMS : UINT := 32;

    // Số conveyor tối đa được khai báo trong hệ thống.
    C_MAX_CONVEYORS : UINT := 2;

    // Giá trị PI kiểu REAL dùng cho các phép đổi góc.
    C_PI : REAL := 3.141592654;
	
	// Hệ số chuyển đổi từ độ sang radian.
    C_DEG_TO_RAD : REAL := 0.01745329252;

    // Hệ số chuyển đổi từ radian sang độ.
    C_RAD_TO_DEG : REAL := 57.29577951;

    // Giá trị rất nhỏ dùng để tránh phép chia cho 0.
    C_REAL_EPSILON : REAL := 0.000001;
	
	C_EPSILON : REAL := 0.000001;

    // Giá trị mặc định dùng để đánh dấu index không hợp lệ.
    C_INVALID_INDEX : UINT := 0;
	
	// So sensor source lon nhat
	C_MAX_SENSOR_SOURCES :UINT := 4;
	// So recipe lon nhat
	C_MAX_TRACK_RECIPES :UINT := 4;
	// Số Vision Source tối đa.
	C_MAX_VISION_SOURCES : UINT := 4;
	
	// Số Object tối đa Vision được phép trả trong một lần chụp.
		
	C_MAX_VISION_TRACK_OBJECTS_PER_FRAME : UINT := 20;
	C_VISION_TRACK_OBJECT_REG_COUNT : UINT := 9;
	C_VISION_TRACK_OBJECTS_PER_BLOCK : UINT := 10;
	C_MAX_VISION_ALIGN_ITERATIONS : UINT := 4;
	C_MAX_VISION_ALIGN_RECIPES : UINT := 16;
	C_MAX_TRAYS : UINT := 16;
		
	C_VISION_CAMERA_REGISTER_SIZE : UINT := 300;
	C_VISION_R2V_REGISTER_COUNT : UINT := 100;
	C_VISION_V2R_REGISTER_COUNT : UINT := 200;
	C_VISION_STATUS_OFFSET : UINT := 100;
	C_VISION_HEADER_OFFSET : UINT := 101;
	C_VISION_SIMPLE_DATA_OFFSET : UINT := 116;
	C_VISION_MULTI_DATA_OFFSET : UINT := 132;
	

	
END_VAR
VAR_GLOBAL
    // Cấu hình các camera.
    g_aVisionConfig :
        ARRAY[0..C_MAX_VISION_CHANNELS] OF ST_VISION_CONFIG;

    // Cấu hình các job vision.
    g_aVisionJobConfig :
        ARRAY[0..C_MAX_VISION_JOBS] OF ST_VISION_JOB_CONFIG;

    // Lệnh gửi tới từng camera.
    g_aVisionCommand :
        ARRAY[0..C_MAX_VISION_CHANNELS] OF ST_VISION_COMMAND;

    // Trạng thái từng camera.
    g_aVisionStatus :
        ARRAY[0..C_MAX_VISION_CHANNELS] OF ST_VISION_CHANNEL_STATUS;

    // Kết quả của từng camera.
    g_aVisionResult :
        ARRAY[0..C_MAX_VISION_CHANNELS] OF ST_VISION_RESULT;
		
	// Monitor Bit Vision
	g_aVision_ControlWord : ARRAY[0..C_MAX_VISION_CHANNELS] OF ST_ControlWord_VS;
	g_aVision_StatusWord : ARRAY[0..C_MAX_VISION_CHANNELS] OF ST_StatusWord_VS;
	
    // Dữ liệu ứng dụng.
    g_stAlignRuntime         : ST_ALIGN_RUNTIME;
    g_stInspectionRuntime    : ST_INSPECTION_RUNTIME;
    g_stGlueRuntime          : ST_GLUE_RUNTIME;

    // Dữ liệu conveyor.
    g_aConveyorRuntime :
        ARRAY[0..C_MAX_CONVEYORS] OF ST_CONVEYOR_RUNTIME;

    // Hàng đợi sản phẩm tracking.
    g_stTrackingQueue_A        : ST_TRACKING_QUEUE;

    // Cấu hình và runtime tracking.
    g_stTrackingConfig_A       : ST_TRACKING_CONFIG;
    g_stTrackingRuntime_A      : ST_TRACKING_RUNTIME;

    // Giai đoạn kiểm thử đang được chọn.
    g_eSystemTestStage       : E_SystemTestStage;
	// Khai bao bien goc cho he toa do Conveyor
	//g_stConveyorOrigin 		 : ST_POS; 
END_VAR
// Application Variable
VAR_GLOBAL
    // Command/response chung giữa Interpreter và Application Manager.
    g_stApplicationCommandA : ST_APPLICATION_COMMAND;
    g_stApplicationResponseA : ST_APPLICATION_RESPONSE;

    // Cấu hình mô phỏng Conveyor Tracking.
    g_stTrackingSimulation : ST_TRACKING_SIMULATION_CONFIG;

    // Quyền sở hữu Motion Queue.
    g_xApplicationMotionOwnerA : BOOL;

    // Adapter tracking → Motion Queue.
    g_xTrackingMotionAccepted : BOOL;
    g_xTrackingMotionBusy : BOOL;
    g_xTrackingMotionDone : BOOL;
    g_xTrackingMotionError : BOOL;
    g_udiTrackingMotionErrorID : UDINT;
    g_xTrackingMotionAbortDone : BOOL;

    // IO logic; sau này map sang IO thật theo Tracking Config.
    g_xTrackingVacuumOutput : BOOL;
    g_xTrackingBlowOutput : BOOL;
    g_xTrackingVacuumOK : BOOL;

    // Recipe tracking. Giai đoạn đầu dùng 1 recipe.
    // Sau khi HMI hoàn thiện có thể đổi thành ARRAY recipe.
    g_xTrackingConfigInitialized : BOOL;
	
	
	// Command từ Interpreter tới Tracking Engine.
    A_TrackStartCmd : BOOL;
    A_TrackAbortCmd : BOOL;
    A_TrackResetCmd : BOOL;

    // Response từ Tracking Engine về Interpreter/HMI.
    A_TrackEngineAccepted : BOOL;
    A_TrackEngineBusy : BOOL;
    A_TrackEngineDone : BOOL;
    A_TrackEngineError : BOOL;
    A_TrackEngineErrorID : UDINT;
    A_TrackEngineState : INT;

END_VAR

VAR_GLOBAL CONSTANT
    // Số lượng Tool tối đa trên một Robot.
    C_MAX_TOOLS : UINT := 8;

    // Số lượng Digital Input logic tối đa.
    C_MAX_DI : UINT := 128;

    // Số lượng Digital Output logic tối đa.
    C_MAX_DO : UINT := 128;

END_VAR

//=============================================================================
// GVL: LOGICAL IO - ROBOT A
//-----------------------------------------------------------------------------
// IO vật lý nên được Map vào các mảng này tại một chương trình riêng.
//=============================================================================
VAR_GLOBAL

    // Command và Status của lệnh TRACK_ON.
	g_stMultiTrackCommandA : ST_MultiToolTrackingCommand;
	g_stMultiTrackStatusA : ST_MultiToolTrackingStatus;
	
	// Cấu hình và Runtime Tool Robot A.
	g_aToolConfigA : ARRAY[0..C_MAX_TOOLS] OF ST_ToolConfig;
	g_aToolStatusA : ARRAY[0..C_MAX_TOOLS] OF ST_ToolStatus;
	
	// Recipe và Queue Robot A.
	g_aMultiTrackRecipeA : ARRAY[0..C_MAX_TRACK_RECIPES] OF ST_MultiToolTrackingRecipe;
	g_stTrackingObjectQueueA : ST_TrackingObjectQueue;
	
	// Cấu hình các nguồn Sensor.
    g_aSensorSourceConfigA : ARRAY[0..C_MAX_SENSOR_SOURCES] OF ST_SensorObjectSourceConfig;

  	// Cấu hình Vision Tracking cho từng Camera/Channel.
	g_aVisionTrackingSourceConfigA : ARRAY[0..C_MAX_VISION_CHANNELS] OF ST_VisionTrackingSourceConfig;
	
	// Multi-object result dành riêng cho Conveyor Tracking.
	g_aVisionTrackingMultiResultA : ARRAY[0..C_MAX_VISION_CHANNELS] OF ST_VisionTrackingMultiResult;
	
	g_aVisionAlignRecipeA : ARRAY[0..C_MAX_VISION_ALIGN_RECIPES] OF ST_VisionAlignRecipe;
	g_aVisionAlignRuntimeA : ARRAY[1..C_MAX_TOOLS] OF ST_VisionAlignToolRuntime;
	g_aTrayConfigA : ARRAY[0..C_MAX_TRAYS] OF ST_TrayConfig;
	g_aTrayRuntimeA : ARRAY[0..C_MAX_TRAYS] OF ST_TrayRuntime;

	
	// Giao tiếp giữa MultiTool Controller và Tracking Core hiện tại.
	g_xMultiTrackCoreExecuteA : BOOL;
	g_xMultiTrackCoreResetA : BOOL;
	g_xMultiTrackCoreAbortA : BOOL;
	g_xMultiTrackPickerSafeA : BOOL;
	
	g_uiMultiTrackObjectIndexA : UINT;
	g_uiMultiTrackToolIDA : UINT;
	g_stMultiTrackPickOffsetA : ST_POS;
	g_rMultiTrackApproachHeightA : REAL;
	
	// Phản hồi từ Tracking Core về MultiTool Controller.
	g_xTrackingCoreAcceptedA : BOOL;
	g_xTrackingCoreBusyA : BOOL;
	g_xTrackingCoreSyncOKA : BOOL;
	g_xTrackingCorePCSInUseA : BOOL;
	g_xTrackingCoreReleasedA : BOOL;
	g_xTrackingCoreErrorA : BOOL;
	g_udiTrackingCoreErrorIDA : UDINT;
	
	// Command Tool được Controller phát ra.
	g_stToolCommandA : ST_ToolCommand;
	
	// Chọn Tool/TCP Robot A.
	g_xSelectToolExecuteA : BOOL;
	g_uiSelectToolIDA : UINT;
	g_stSelectToolTCPA : ST_POS;
	g_xSelectToolDoneA : BOOL;
	g_xSelectToolErrorA : BOOL;
	g_udiSelectToolErrorIDA : UDINT;
	
	// IO logic Tool Robot A.
	// Nếu project đã có mảng IO chung thì dùng mảng cũ và không khai báo lại.
	g_axDIA : ARRAY[0..C_MAX_DI] OF BOOL;
	g_axDORequestToolA : ARRAY[0..C_MAX_DO] OF BOOL;
	
	// Bit test commissioning. Không dùng trong Interpreter chính thức.
	g_xMultiTrackStartTestA : BOOL;
	g_xMultiTrackResetTestA : BOOL;
	g_xMultiTrackAbortTestA : BOOL;
	g_xCreateTestTrackingObjectA : BOOL;
	
	// TRUE khi cấu hình Multi-tool Robot A đã được khởi tạo.
	g_xMultiToolConfigInitializedA : BOOL := FALSE;
	
	// Bit cho phép khởi tạo lại giá trị mặc định khi commissioning.
	g_xInitializeMultiToolConfigA : BOOL := FALSE;
	
	g_xClearTrackingQueueA : BOOL;
	g_xResetTrackingObjectSourceA : BOOL;
	
	//=============================================================================
	// TRACKING APPLICATION RESULT - ROBOT A
	//=============================================================================
	g_xTrackOKA : BOOL;              // TRUE khi lệnh Tracking gần nhất Pick đủ số lượng.
	g_xTrackErrorA : BOOL;           // TRUE khi lệnh Tracking kết thúc lỗi.
	g_udiTrackErrorIDA : UDINT;      // ErrorID của lệnh Tracking gần nhất.
	g_udiTrackDoneCommandIDA : UDINT;// CommandID đã hoàn thành.
	//=============================================================================
	// TOOL COMMAND TỪ INTERPRETER - ROBOT A
	//=============================================================================
	g_stInterpreterToolCommandA : ST_ToolCommand;
	
	g_HMI_PulsePerCycle_Cr: REAL;
	g_HMI_PulsePerCycle_Set : INT;
	
	// Cho phép test Background Vision Trigger mà chưa cần chạy TRACK_PICK.
	// Production bình thường phải để FALSE.
	g_xVisionTrackingAutoTriggerTestA : BOOL := FALSE;

END_VAR

//=============================================================================
// GVL_HMI_TOOL_CONFIG
//-----------------------------------------------------------------------------
// Biến trung gian phục vụ màn hình cấu hình Tool dùng chung cho Robot A và B.
//=============================================================================
VAR_GLOBAL

    //=========================================================================
    // ROBOT A
    //=========================================================================

    // Dữ liệu chỉnh sửa Tool Robot A.
    g_stHMIToolEditorA : ST_HMIToolConfigEditor;

    // Trạng thái Tool đang được chọn của Robot A.
    // HMI chỉ đọc biến này, không ghi trực tiếp vào mảng ToolStatus.
    g_stHMIToolStatusA : ST_ToolStatus;

    // Các bộ bắt cạnh lệnh HMI Robot A.
    g_rtHMIToolLoadA : R_TRIG;
    g_rtHMIToolSaveA : R_TRIG;
    g_rtHMIToolCancelA : R_TRIG;

    // Index Tool được chọn ở vòng quét trước.
    g_uiHMIToolSelectedIndexOldA : UINT;

    // Biến chạy vòng FOR kiểm tra ToolID trùng.
    g_uiHMIToolCheckIndexA : UINT;

    // TRUE khi phát hiện ToolID bị trùng.
    g_xHMIToolDuplicateIDA : BOOL;


    //=========================================================================
    // ROBOT B
    //=========================================================================

    // Dữ liệu chỉnh sửa Tool Robot B.
    g_stHMIToolEditorB : ST_HMIToolConfigEditor;

    // Trạng thái Tool đang được chọn của Robot B.
    g_stHMIToolStatusB : ST_ToolStatus;

    // Các bộ bắt cạnh lệnh HMI Robot B.
    g_rtHMIToolLoadB : R_TRIG;
    g_rtHMIToolSaveB : R_TRIG;
    g_rtHMIToolCancelB : R_TRIG;

    // Index Tool được chọn ở vòng quét trước.
    g_uiHMIToolSelectedIndexOldB : UINT;

    // Biến chạy vòng FOR kiểm tra ToolID trùng.
    g_uiHMIToolCheckIndexB : UINT;

    // TRUE khi phát hiện ToolID bị trùng.
    g_xHMIToolDuplicateIDB : BOOL;

END_VAR

//=============================================================================
// GVL_HMI_TOOL_CONFIG
//-----------------------------------------------------------------------------
// Biến trung gian phục vụ màn hình cấu hình Tool dùng chung cho Robot A và B.
//=============================================================================

VAR_GLOBAL
	g_stHMIConveyor_Config_Save: BOOL;
	g_stHMITracking_Config_Save: BOOL;
	g_stHMIConveyor_Config_Read: BOOL;
	g_stHMITracking_Config_Read: BOOL;
	g_stHMITool_Config_Read_All: BOOL;
	g_stHMITool_Config_Save_All: BOOL;
END_VAR

//=============================================================================
// GVL_HMI_SENSOR SOURCE_CONFIG
//-----------------------------------------------------------------------------
// Biến trung gian phục vụ màn hình cấu hình sensor source dùng chung cho Robot A.
//====
VAR_GLOBAL
	// Sensor Source đang chọn trên HMI.
	g_uiHMISensorSourceIndexA : UINT := 1;
	
	// Dữ liệu trung gian HMI.
	g_stHMISensorSourceA : ST_SensorObjectSourceConfig;
	
	// Lệnh HMI.
	g_xHMILoadSensorSourceA : BOOL;
	g_xHMISaveSensorSourceA : BOOL;
	g_xHMILoadSensorSourceA_All: BOOL;
	g_xHMISaveSensorSourceA_All : BOOL;
END_VAR

//=============================================================================
// GVL_HMI_RECIPE_CONFIG
//-----------------------------------------------------------------------------
// Biến trung gian phục vụ màn hình cấu hình recipe dùng chung cho Robot A.
//====
VAR_GLOBAL
	// Recipe đang chọn trên HMI.
	g_uiHMITrackingRecipeIndexA : UINT := 1;
	// Dữ liệu trung gian HMI.
	g_stHMITrackingRecipeA : ST_MultiToolTrackingRecipe;
	// Lệnh HMI.
	g_xHMILoadTrackingRecipeA : BOOL;
	g_xHMISaveTrackingRecipeA : BOOL;
	g_xHMILoadTrackingRecipeA_All : BOOL;
	g_xHMISaveTrackingRecipeA_All : BOOL;
END_VAR

//=============================================================================
// GVL_HMI_VISION_SOURCE
//-----------------------------------------------------------------------------
// Biến trung gian phục vụ màn hình cấu hình vision source dùng chung cho Robot A.
//====
VAR_GLOBAL
	g_uiHMIVisionSourceIndexA : UINT := 1;

	g_stHMIVisionSourceA : ST_VisionTrackingSourceConfig;
	
	g_xHMILoadVisionSourceA : BOOL;
	g_xHMISaveVisionSourceA : BOOL;
	g_xHMISaveAllVisionSourceA : BOOL;
	g_xHMILoadAllVisionSourceA : BOOL := FALSE;
	
	//=============================================================================
	// ROBOT A - LAST VISION ALIGN RESULT
	//=============================================================================
	A_VisionHeaderOK : BOOL;                    // Header của Result cuối hợp lệ.
	A_VisionTriggerID : UDINT;                  // TriggerID cuối cùng.
	
	A_VisionX : REAL;                           // X Vision trả về.
	A_VisionY : REAL;                           // Y Vision trả về.
	A_VisionZ : REAL;                           // Z Vision trả về.
	A_VisionA : REAL;                           // Góc Vision trả về.
	A_VisionScore : REAL;                       // Score Vision.
	A_VisionFeatureID : UINT;                   // FeatureID Vision.

END_VAR

// VISION MODBUS

VAR_GLOBAL
	g_aVisionModbusControl : ARRAY[0..C_MAX_VISION_CHANNELS] OF ST_VISION_MODBUS_CONTROL;
	g_aVisionModbusStatus : ARRAY[0..C_MAX_VISION_CHANNELS] OF ST_VISION_MODBUS_STATUS;
END_VAR

VAR_GLOBAL
	//=============================================================================
	// 1. THÊM VÀO GVL
	//=============================================================================
	
	// Mỗi lần cần Apply lại Tool/TCP thì tăng RequestID.
	g_udiRobotAToolApplyRequestA : UDINT := 0;
	
	// RequestID đã Apply thành công.
	g_udiRobotAToolAppliedRequestA : UDINT := 0;
	
	// Trạng thái Apply Tool.
	g_xRobotAToolApplyBusy : BOOL := FALSE;
	g_xRobotAToolApplyDone : BOOL := FALSE;
	g_xRobotAToolApplyError : BOOL := FALSE;
	g_udiRobotAToolApplyErrorID : UDINT := 0;

END_VAR

// ------------------------------
// ROBOT B
// ------------------------------
// ROBOT B - add these variables into GVL
// Generated from Robot A variables actually used by current Interpreter/MotionManager

VAR_GLOBAL
	B_ActiveMotionCount : INT;
	B_CallStack : ARRAY[0..20] OF INT;
	B_CallStackIndex : INT;
	B_CurrentMotionParam : ST_MotionParam := (Speed := 500.0, Acc := 2000.0, Dec := 2000.0, Jerk := 10000.0, VelFac := 1.0, AccFac := 1.0, DecFac := 1.0, JerkFac := 1.0);
	B_LastStepRunReq : BOOL;
	B_LengthStep : INT;
	B_MotionAbortDone : BOOL;
	B_MotionAbortReq : BOOL;
	B_MotionCount : INT := 0;
	B_MotionDonePulse : BOOL;
	B_MotionDoneStep : INT;
	B_MotionErrorCode : INT;
	B_MotionErrorPulse : BOOL;
	B_MotionErrorSlot : INT;
	B_MotionErrorStep : INT;
	B_MotionQueue : ARRAY[0..20] OF ST_MotionQueueItem;
	B_MotionHead : INT := 1;
	B_MotionManagerBusy : BOOL;
	B_MotionManagerDone : BOOL;
	B_MotionManagerError : BOOL;
	B_MotionManagerState : INT;
	B_MotionTail : INT := 1;
	B_MoveSlotAccepted : ARRAY[0..3] OF BOOL;
	B_MoveSlotBusy : ARRAY[0..3] OF BOOL;
	B_MoveSlotCmd : ARRAY[0..3] OF E_RobotCmd;
	B_MoveSlotDone : ARRAY[0..3] OF BOOL;
	B_MoveSlotError : ARRAY[0..3] OF BOOL;
	B_MoveSlotErrorID : ARRAY[0..3] OF INT;
	B_MoveSlotItem : ARRAY[0..3] OF ST_MotionQueueItem;
	B_MoveSlotReleasePending : ARRAY[0..3] OF BOOL;
	B_MoveSlotStart : ARRAY[0..3] OF BOOL;
	B_PipelineActive : BOOL;
	B_PipelineDepth : INT := 3;
	B_PipelineNextPushStep : INT;
	B_PipelineUsedCount : INT := 0;
	B_PushMotionDone : BOOL;
	B_PushMotionError : BOOL;
	B_PushMotionItem : ST_MotionQueueItem;
	B_PushMotionReq : BOOL;
	B_Reg : ARRAY[0..200] OF DINT;
	B_RunAlarm : BOOL;
	B_RunAlarmCode : INT;
	B_RunBusy : BOOL;
	B_RunDone : BOOL;
	B_RunEnable : BOOL;
	B_RunErrorStep : INT;
	B_RunMode : INT := 0;
	B_RunPause : BOOL;
	B_RunState : INT := 0;
	B_RunStep : INT := 1;
	B_RunStop : BOOL;
	B_StepActive : BOOL;
	B_StepHold : BOOL;
	B_StepRunEdge : BOOL;
	B_StepRunReq : BOOL;
	B_TimerDone : ARRAY[0..20] OF BOOL;
	B_TimerPT : ARRAY[0..20] OF TIME;
	B_TimerStart : ARRAY[0..20] OF BOOL;
	B_TrackEnable : BOOL;
	B_TrackEngineBusy : BOOL;
	B_TrackEngineDone : BOOL;
	B_TrackEngineError : BOOL;
	B_TrackEngineErrorID : UDINT;
	B_TrackPlaceDone : BOOL;
	B_TrackPlaceReq : BOOL;
	B_TrackStartCmd : BOOL;
	B_Var : ARRAY[0..200] OF DINT;
	B_VisionDone : BOOL;
	B_VisionError : BOOL;
	B_VisionOK : BOOL;
	B_VisionTriggerReq : BOOL;
END_VAR

